METHOD Create : RTS_IEC_HANDLE
  VAR_INPUT
    iAddressFamily : INT;  (* Socket address family *)
    diType : DINT;  (* Socket TYPE *)
    diProtocol : DINT;  (* Socket protocol *)
    pResult : POINTER TO RTS_IEC_RESULT;  (* Pointer to runtime system error code (see CmpErrors.library) *)
  END_VAR
                          // check, for reinitilaization
IF (THIS^.hSocket = RTS_INVALID_HANDLE) THEN
	THIS^.hSocket := SysSocket.SysSockCreate(iAddressFamily, diType, diProtocol, pResult);
	Create := THIS^.hSocket;
ELSE
	Create := RTS_INVALID_HANDLE;
END_IF
                        
END_METHOD
END_FUNCTION_BLOCK

FUNCTION_BLOCK _FB_ETHRx_Message_Unpack
  VAR_INPUT
    I_Byte_0 : BYTE;
    I_Byte_1 : BYTE;
    I_Byte_2 : BYTE;
    I_Byte_3 : BYTE;
    I_Byte_4 : BYTE;
    I_Byte_5 : BYTE;
    I_Byte_6 : BYTE;
    I_Byte_7 : BYTE;
  END_VAR
  VAR_OUTPUT
    S_ER_TmOut : BOOL;  (* Input data endpoints *)
    S_Bit_0 : BOOL;  (* Input data endpoints *)
    S_Bit_1 : BOOL;  (* Input data endpoints *)
    S_Bit_2 : BOOL;  (* Input data endpoints *)
    S_Bit_3 : BOOL;  (* Input data endpoints *)
    S_Bit_4 : BOOL;  (* Input data endpoints *)
    S_Bit_5 : BOOL;  (* Input data endpoints *)
    S_Bit_6 : BOOL;  (* Input data endpoints *)
    S_Bit_7 : BOOL;  (* Input data endpoints *)
    X_Byte_0 : BYTE;  (* Input data endpoints *)
    S_Bit_8 : BOOL;  (* Input data endpoints *)
    S_Bit_9 : BOOL;  (* Input data endpoints *)
    S_Bit_10 : BOOL;  (* Input data endpoints *)
    S_Bit_11 : BOOL;  (* Input data endpoints *)
    S_Bit_12 : BOOL;  (* Input data endpoints *)
    S_Bit_13 : BOOL;  (* Input data endpoints *)
    S_Bit_14 : BOOL;  (* Input data endpoints *)
    S_Bit_15 : BOOL;  (* Input data endpoints *)
    X_Byte_1 : BYTE;  (* Input data endpoints *)
    X_Word_0 : WORD;  (* Input data endpoints *)
    S_Bit_16 : BOOL;  (* Input data endpoints *)
    S_Bit_17 : BOOL;  (* Input data endpoints *)
    S_Bit_18 : BOOL;  (* Input data endpoints *)
    S_Bit_19 : BOOL;  (* Input data endpoints *)
    S_Bit_20 : BOOL;  (* Input data endpoints *)
    S_Bit_21 : BOOL;  (* Input data endpoints *)
    S_Bit_22 : BOOL;  (* Input data endpoints *)
    S_Bit_23 : BOOL;  (* Input data endpoints *)
    X_Byte_2 : BYTE;  (* Input data endpoints *)
    S_Bit_24 : BOOL;  (* Input data endpoints *)
    S_Bit_25 : BOOL;  (* Input data endpoints *)
    S_Bit_26 : BOOL;  (* Input data endpoints *)
    S_Bit_27 : BOOL;  (* Input data endpoints *)
    S_Bit_28 : BOOL;  (* Input data endpoints *)
    S_Bit_29 : BOOL;  (* Input data endpoints *)
    S_Bit_30 : BOOL;  (* Input data endpoints *)
    S_Bit_31 : BOOL;  (* Input data endpoints *)
    X_Byte_3 : BYTE;  (* Input data endpoints *)
    S_Bit_32 : BOOL;  (* Input data endpoints *)
    S_Bit_33 : BOOL;  (* Input data endpoints *)
    S_Bit_34 : BOOL;  (* Input data endpoints *)
    S_Bit_35 : BOOL;  (* Input data endpoints *)
    S_Bit_36 : BOOL;  (* Input data endpoints *)
    S_Bit_37 : BOOL;  (* Input data endpoints *)
    S_Bit_38 : BOOL;  (* Input data endpoints *)
    S_Bit_39 : BOOL;  (* Input data endpoints *)
    X_Byte_4 : BYTE;  (* Input data endpoints *)
    S_Bit_40 : BOOL;  (* Input data endpoints *)
    S_Bit_41 : BOOL;  (* Input data endpoints *)
    S_Bit_42 : BOOL;  (* Input data endpoints *)
    S_Bit_43 : BOOL;  (* Input data endpoints *)
    S_Bit_44 : BOOL;  (* Input data endpoints *)
    S_Bit_45 : BOOL;  (* Input data endpoints *)
    S_Bit_46 : BOOL;  (* Input data endpoints *)
    S_Bit_47 : BOOL;  (* Input data endpoints *)
    X_Byte_5 : BYTE;  (* Input data endpoints *)
    X_Word_2 : WORD;  (* Input data endpoints *)
    S_Bit_48 : BOOL;  (* Input data endpoints *)
    S_Bit_49 : BOOL;  (* Input data endpoints *)
    S_Bit_50 : BOOL;  (* Input data endpoints *)
    S_Bit_51 : BOOL;  (* Input data endpoints *)
    S_Bit_52 : BOOL;  (* Input data endpoints *)
    S_Bit_53 : BOOL;  (* Input data endpoints *)
    S_Bit_54 : BOOL;  (* Input data endpoints *)
    S_Bit_55 : BOOL;  (* Input data endpoints *)
    X_Byte_6 : BYTE;  (* Input data endpoints *)
    S_Bit_56 : BOOL;  (* Input data endpoints *)
    S_Bit_57 : BOOL;  (* Input data endpoints *)
    S_Bit_58 : BOOL;  (* Input data endpoints *)
    S_Bit_59 : BOOL;  (* Input data endpoints *)
    S_Bit_60 : BOOL;  (* Input data endpoints *)
    S_Bit_61 : BOOL;  (* Input data endpoints *)
    S_Bit_62 : BOOL;  (* Input data endpoints *)
    S_Bit_63 : BOOL;  (* Input data endpoints *)
    X_Byte_7 : BYTE;  (* Input data endpoints *)
  END_VAR

                    			X_Byte_0 :=I_Byte_0;			
            X_Byte_1 :=I_Byte_1;
            X_Byte_2 :=I_Byte_2;
            X_Byte_3 :=I_Byte_3;
            X_Byte_4 :=I_Byte_4;
            X_Byte_5 :=I_Byte_5;
			X_Byte_6 :=I_Byte_6;
            X_Byte_7 :=I_Byte_7;
			
			S_Bit_0  := BYTE_TO_BOOL(X_Byte_0 AND 2#00000001);
			S_Bit_1  := BYTE_TO_BOOL(X_Byte_0 AND 2#00000010);
			S_Bit_2  := BYTE_TO_BOOL(X_Byte_0 AND 2#00000100);
			S_Bit_3  := BYTE_TO_BOOL(X_Byte_0 AND 2#00001000);
			S_Bit_4  := BYTE_TO_BOOL(X_Byte_0 AND 2#00010000);
			S_Bit_5  := BYTE_TO_BOOL(X_Byte_0 AND 2#00100000);
			S_Bit_6  := BYTE_TO_BOOL(X_Byte_0 AND 2#01000000);
			S_Bit_7  := BYTE_TO_BOOL(X_Byte_0 AND 2#10000000);
			S_Bit_8  := BYTE_TO_BOOL(X_Byte_1 AND 2#00000001);
			S_Bit_9  := BYTE_TO_BOOL(X_Byte_1 AND 2#00000010);
			S_Bit_10  := BYTE_TO_BOOL(X_Byte_1 AND 2#00000100);
			S_Bit_11  := BYTE_TO_BOOL(X_Byte_1 AND 2#00001000);
			S_Bit_12  := BYTE_TO_BOOL(X_Byte_1 AND 2#00010000);
			S_Bit_13  := BYTE_TO_BOOL(X_Byte_1 AND 2#00100000);
			S_Bit_14  := BYTE_TO_BOOL(X_Byte_1 AND 2#01000000);
			S_Bit_15  := BYTE_TO_BOOL(X_Byte_1 AND 2#10000000);
			S_Bit_16  := BYTE_TO_BOOL(X_Byte_2 AND 2#00000001);
			S_Bit_17  := BYTE_TO_BOOL(X_Byte_2 AND 2#00000010);
			S_Bit_18  := BYTE_TO_BOOL(X_Byte_2 AND 2#00000100);
			S_Bit_19  := BYTE_TO_BOOL(X_Byte_2 AND 2#00001000);
			S_Bit_20  := BYTE_TO_BOOL(X_Byte_2 AND 2#00010000);
			S_Bit_21  := BYTE_TO_BOOL(X_Byte_2 AND 2#00100000);
			S_Bit_22  := BYTE_TO_BOOL(X_Byte_2 AND 2#01000000);
			S_Bit_23  := BYTE_TO_BOOL(X_Byte_2 AND 2#10000000);
			S_Bit_24  := BYTE_TO_BOOL(X_Byte_3 AND 2#00000001);
			S_Bit_25  := BYTE_TO_BOOL(X_Byte_3 AND 2#00000010);
			S_Bit_26  := BYTE_TO_BOOL(X_Byte_3 AND 2#00000100);
			S_Bit_27  := BYTE_TO_BOOL(X_Byte_3 AND 2#00001000);
			S_Bit_28  := BYTE_TO_BOOL(X_Byte_3 AND 2#00010000);
			S_Bit_29  := BYTE_TO_BOOL(X_Byte_3 AND 2#00100000);
			S_Bit_30  := BYTE_TO_BOOL(X_Byte_3 AND 2#01000000);
			S_Bit_31  := BYTE_TO_BOOL(X_Byte_3 AND 2#10000000);
			S_Bit_32  := BYTE_TO_BOOL(X_Byte_4 AND 2#00000001);
			S_Bit_33  := BYTE_TO_BOOL(X_Byte_4 AND 2#00000010);
			S_Bit_34  := BYTE_TO_BOOL(X_Byte_4 AND 2#00000100);
			S_Bit_35  := BYTE_TO_BOOL(X_Byte_4 AND 2#00001000);
			S_Bit_36  := BYTE_TO_BOOL(X_Byte_4 AND 2#00010000);
			S_Bit_37  := BYTE_TO_BOOL(X_Byte_4 AND 2#00100000);
			S_Bit_38  := BYTE_TO_BOOL(X_Byte_4 AND 2#01000000);
			S_Bit_39  := BYTE_TO_BOOL(X_Byte_4 AND 2#10000000);
			S_Bit_40  := BYTE_TO_BOOL(X_Byte_5 AND 2#00000001);
			S_Bit_41  := BYTE_TO_BOOL(X_Byte_5 AND 2#00000010);
			S_Bit_42  := BYTE_TO_BOOL(X_Byte_5 AND 2#00000100);
			S_Bit_43  := BYTE_TO_BOOL(X_Byte_5 AND 2#00001000);
			S_Bit_44  := BYTE_TO_BOOL(X_Byte_5 AND 2#00010000);
			S_Bit_45  := BYTE_TO_BOOL(X_Byte_5 AND 2#00100000);
			S_Bit_46  := BYTE_TO_BOOL(X_Byte_5 AND 2#01000000);
			S_Bit_47  := BYTE_TO_BOOL(X_Byte_5 AND 2#10000000);
			S_Bit_48  := BYTE_TO_BOOL(X_Byte_6 AND 2#00000001);
			S_Bit_49  := BYTE_TO_BOOL(X_Byte_6 AND 2#00000010);
			S_Bit_50  := BYTE_TO_BOOL(X_Byte_6 AND 2#00000100);
			S_Bit_51  := BYTE_TO_BOOL(X_Byte_6 AND 2#00001000);
			S_Bit_52  := BYTE_TO_BOOL(X_Byte_6 AND 2#00010000);
			S_Bit_53  := BYTE_TO_BOOL(X_Byte_6 AND 2#00100000);
			S_Bit_54  := BYTE_TO_BOOL(X_Byte_6 AND 2#01000000);
			S_Bit_55  := BYTE_TO_BOOL(X_Byte_6 AND 2#10000000);
			S_Bit_56  := BYTE_TO_BOOL(X_Byte_7 AND 2#00000001);
			S_Bit_57  := BYTE_TO_BOOL(X_Byte_7 AND 2#00000010);
			S_Bit_58  := BYTE_TO_BOOL(X_Byte_7 AND 2#00000100);
			S_Bit_59  := BYTE_TO_BOOL(X_Byte_7 AND 2#00001000);
			S_Bit_60  := BYTE_TO_BOOL(X_Byte_7 AND 2#00010000);
			S_Bit_61  := BYTE_TO_BOOL(X_Byte_7 AND 2#00100000);
			S_Bit_62  := BYTE_TO_BOOL(X_Byte_7 AND 2#01000000);
			S_Bit_63  := BYTE_TO_BOOL(X_Byte_7 AND 2#10000000);
                  
END_FUNCTION_BLOCK

FUNCTION_BLOCK _FB_ETHTx_Message_Unpack
  VAR_INPUT
    S_Bit_0 : BOOL := FALSE;  (* Message Datas *)
    S_Bit_1 : BOOL := FALSE;  (* Message Datas *)
    S_Bit_2 : BOOL := FALSE;  (* Message Datas *)
    S_Bit_3 : BOOL := FALSE;  (* Message Datas *)
    S_Bit_4 : BOOL := FALSE;  (* Message Datas *)
    S_Bit_5 : BOOL := FALSE;  (* Message Datas *)
    S_Bit_6 : BOOL := FALSE;  (* Message Datas *)
    S_Bit_7 : BOOL := FALSE;  (* Message Datas *)
    X_Byte_0 : BYTE := 16#0;  (* Message Datas *)
    S_Bit_8 : BOOL := FALSE;  (* Message Datas *)
    S_Bit_9 : BOOL := FALSE;  (* Message Datas *)
    S_Bit_10 : BOOL := FALSE;  (* Message Datas *)
    S_Bit_11 : BOOL := FALSE;  (* Message Datas *)
    S_Bit_12 : BOOL := FALSE;  (* Message Datas *)
    S_Bit_13 : BOOL := FALSE;  (* Message Datas *)
    S_Bit_14 : BOOL := FALSE;  (* Message Datas *)
    S_Bit_15 : BOOL := FALSE;  (* Message Datas *)
    X_Byte_1 : BYTE := 16#0;  (* Message Datas *)
    S_Bit_16 : BOOL := FALSE;  (* Message Datas *)
    S_Bit_17 : BOOL := FALSE;  (* Message Datas *)
    S_Bit_18 : BOOL := FALSE;  (* Message Datas *)
    S_Bit_19 : BOOL := FALSE;  (* Message Datas *)
    S_Bit_20 : BOOL := FALSE;  (* Message Datas *)
    S_Bit_21 : BOOL := FALSE;  (* Message Datas *)
    S_Bit_22 : BOOL := FALSE;  (* Message Datas *)
    S_Bit_23 : BOOL := FALSE;  (* Message Datas *)
    X_Byte_2 : BYTE := 16#0;  (* Message Datas *)
    S_Bit_24 : BOOL := FALSE;  (* Message Datas *)
    S_Bit_25 : BOOL := FALSE;  (* Message Datas *)
    S_Bit_26 : BOOL := FALSE;  (* Message Datas *)
    S_Bit_27 : BOOL := FALSE;  (* Message Datas *)
    S_Bit_28 : BOOL := FALSE;  (* Message Datas *)
    S_Bit_29 : BOOL := FALSE;  (* Message Datas *)
    S_Bit_30 : BOOL := FALSE;  (* Message Datas *)
    S_Bit_31 : BOOL := FALSE;  (* Message Datas *)
    X_Byte_3 : BYTE := 16#0;  (* Message Datas *)
    S_Bit_32 : BOOL := FALSE;  (* Message Datas *)
    S_Bit_33 : BOOL := FALSE;  (* Message Datas *)
    S_Bit_34 : BOOL := FALSE;  (* Message Datas *)
    S_Bit_35 : BOOL := FALSE;  (* Message Datas *)
    S_Bit_36 : BOOL := FALSE;  (* Message Datas *)
    S_Bit_37 : BOOL := FALSE;  (* Message Datas *)
    S_Bit_38 : BOOL := FALSE;  (* Message Datas *)
    S_Bit_39 : BOOL := FALSE;  (* Message Datas *)
    X_Byte_4 : BYTE := 16#0;  (* Message Datas *)
    S_Bit_40 : BOOL := FALSE;  (* Message Datas *)
    S_Bit_41 : BOOL := FALSE;  (* Message Datas *)
    S_Bit_42 : BOOL := FALSE;  (* Message Datas *)
    S_Bit_43 : BOOL := FALSE;  (* Message Datas *)
    S_Bit_44 : BOOL := FALSE;  (* Message Datas *)
    S_Bit_45 : BOOL := FALSE;  (* Message Datas *)
    S_Bit_46 : BOOL := FALSE;  (* Message Datas *)
    S_Bit_47 : BOOL := FALSE;  (* Message Datas *)
    X_Byte_5 : BYTE := 16#0;  (* Message Datas *)
    S_Bit_48 : BOOL := FALSE;  (* Message Datas *)
    S_Bit_49 : BOOL := FALSE;  (* Message Datas *)
    S_Bit_50 : BOOL := FALSE;  (* Message Datas *)
    S_Bit_51 : BOOL := FALSE;  (* Message Datas *)
    S_Bit_52 : BOOL := FALSE;  (* Message Datas *)
    S_Bit_53 : BOOL := FALSE;  (* Message Datas *)
    S_Bit_54 : BOOL := FALSE;  (* Message Datas *)
    S_Bit_55 : BOOL := FALSE;  (* Message Datas *)
    X_Byte_6 : BYTE := 16#0;  (* Message Datas *)
    S_Bit_56 : BOOL := FALSE;  (* Message Datas *)
    S_Bit_57 : BOOL := FALSE;  (* Message Datas *)
    S_Bit_58 : BOOL := FALSE;  (* Message Datas *)
    S_Bit_59 : BOOL := FALSE;  (* Message Datas *)
    S_Bit_60 : BOOL := FALSE;  (* Message Datas *)
    S_Bit_61 : BOOL := FALSE;  (* Message Datas *)
    S_Bit_62 : BOOL := FALSE;  (* Message Datas *)
    S_Bit_63 : BOOL := FALSE;  (* Message Datas *)
    X_Byte_7 : BYTE := 16#0;  (* Message Datas *)
  END_VAR
  VAR_OUTPUT
    O_Byte_0 : BYTE;
    O_Byte_1 : BYTE;
    O_Byte_2 : BYTE;
    O_Byte_3 : BYTE;
    O_Byte_4 : BYTE;
    O_Byte_5 : BYTE;
    O_Byte_6 : BYTE;
    O_Byte_7 : BYTE;
  END_VAR
  VAR
    _FB_Pack_Bit_To_Byte_01 : _FB_PACK_8BITS_TO_BYTE;
    _FB_Pack_Bit_To_Byte_02 : _FB_PACK_8BITS_TO_BYTE;
    _FB_Pack_Bit_To_Byte_03 : _FB_PACK_8BITS_TO_BYTE;
    _FB_Pack_Bit_To_Byte_04 : _FB_PACK_8BITS_TO_BYTE;
    _FB_Pack_Bit_To_Byte_05 : _FB_PACK_8BITS_TO_BYTE;
    _FB_Pack_Bit_To_Byte_06 : _FB_PACK_8BITS_TO_BYTE;
    _FB_Pack_Bit_To_Byte_07 : _FB_PACK_8BITS_TO_BYTE;
    _FB_Pack_Bit_To_Byte_08 : _FB_PACK_8BITS_TO_BYTE;
  END_VAR

                    IF X_Byte_0 <> 0 THEN
	
	O_Byte_0 := X_Byte_0;
	
ELSIF S_Bit_0 OR S_Bit_1 OR S_Bit_2 OR S_Bit_3 OR S_Bit_4 OR S_Bit_5 OR S_Bit_6 OR S_Bit_7 THEN			(*Check the bits, pack and assign to the output data*)
	_FB_Pack_Bit_To_Byte_01(
	S_Bit_0:= S_Bit_0, 
	S_Bit_1:= S_Bit_1, 
	S_Bit_2:= S_Bit_2, 
	S_Bit_3:= S_Bit_3, 
	S_Bit_4:= S_Bit_4, 
	S_Bit_5:= S_Bit_5, 
	S_Bit_6:= S_Bit_6, 
	S_Bit_7:= S_Bit_7, 
	X_Byte_0=> O_Byte_0);
ELSE
	O_Byte_0 := 0;
END_IF
		
IF X_Byte_1 <> 0 THEN
	O_Byte_1 := X_Byte_1;
ELSIF S_Bit_8 OR S_Bit_9 OR S_Bit_10 OR S_Bit_11 OR S_Bit_12 OR S_Bit_13 OR S_Bit_14 OR S_Bit_15 THEN			(*Check the bits, pack and assign to the output data*)
	_FB_Pack_Bit_To_Byte_02(
	S_Bit_0:= S_Bit_8, 
	S_Bit_1:= S_Bit_9, 
	S_Bit_2:= S_Bit_10, 
	S_Bit_3:= S_Bit_11, 
	S_Bit_4:= S_Bit_12, 
	S_Bit_5:= S_Bit_13, 
	S_Bit_6:= S_Bit_14, 
	S_Bit_7:= S_Bit_15, 
	X_Byte_0=> O_Byte_1);
ELSE
	O_Byte_1 :=0;
END_IF
	

IF X_Byte_2 <> 0 THEN
	O_Byte_2 := X_Byte_2;
ELSIF S_Bit_16 OR S_Bit_17 OR S_Bit_18 OR S_Bit_19 OR S_Bit_20 OR S_Bit_21 OR S_Bit_22 OR S_Bit_23 THEN				(*Check the bits, pack and assign to the output data*)
	_FB_Pack_Bit_To_Byte_03(
	S_Bit_0:= S_Bit_16, 
	S_Bit_1:= S_Bit_17, 
	S_Bit_2:= S_Bit_18, 
	S_Bit_3:= S_Bit_19, 
	S_Bit_4:= S_Bit_20, 
	S_Bit_5:= S_Bit_21, 
	S_Bit_6:= S_Bit_22, 
	S_Bit_7:= S_Bit_23, 
	X_Byte_0=> O_Byte_2);
ELSE
	O_Byte_2 :=0;
END_IF
		
IF X_Byte_3 <> 0 THEN
	O_Byte_3 := X_Byte_3;
ELSIF S_Bit_24 OR S_Bit_25 OR S_Bit_26 OR S_Bit_27 OR S_Bit_28 OR S_Bit_29 OR S_Bit_30 OR S_Bit_31 THEN				(*Check the bits, pack and assign to the output data*)
	_FB_Pack_Bit_To_Byte_04(
	S_Bit_0:= S_Bit_24, 
	S_Bit_1:= S_Bit_25, 
	S_Bit_2:= S_Bit_26, 
	S_Bit_3:= S_Bit_27, 
	S_Bit_4:= S_Bit_28, 
	S_Bit_5:= S_Bit_29, 
	S_Bit_6:= S_Bit_30, 
	S_Bit_7:= S_Bit_31, 
	X_Byte_0=> O_Byte_3);
ELSE
	O_Byte_3 :=0;
END_IF



IF X_Byte_4 <> 0 THEN
	O_Byte_4 := X_Byte_4;
ELSIF S_Bit_32 OR S_Bit_33 OR S_Bit_34 OR S_Bit_35 OR S_Bit_36 OR S_Bit_37 OR S_Bit_38 OR S_Bit_39 THEN				(*Check the bits, pack and assign to the output data*)
	_FB_Pack_Bit_To_Byte_05(
	S_Bit_0:= S_Bit_32, 
	S_Bit_1:= S_Bit_33, 
	S_Bit_2:= S_Bit_34, 
	S_Bit_3:= S_Bit_35, 
	S_Bit_4:= S_Bit_36, 
	S_Bit_5:= S_Bit_37, 
	S_Bit_6:= S_Bit_38, 
	S_Bit_7:= S_Bit_39, 
	X_Byte_0=> O_Byte_4);	
ELSE
	O_Byte_4 :=0;
END_IF
		
IF X_Byte_5 <> 0 THEN
	O_Byte_5 := X_Byte_5;
ELSIF S_Bit_40 OR S_Bit_41 OR S_Bit_42 OR S_Bit_43 OR S_Bit_44 OR S_Bit_45 OR S_Bit_46 OR S_Bit_47 THEN				(*Check the bits, pack and assign to the output data*)
	_FB_Pack_Bit_To_Byte_06(
	S_Bit_0:= S_Bit_40, 
	S_Bit_1:= S_Bit_41, 
	S_Bit_2:= S_Bit_42, 
	S_Bit_3:= S_Bit_43, 
	S_Bit_4:= S_Bit_44, 
	S_Bit_5:= S_Bit_45, 
	S_Bit_6:= S_Bit_46, 
	S_Bit_7:= S_Bit_47, 
	X_Byte_0=> O_Byte_5);
ELSE
	O_Byte_5 :=0;
END_IF

	

IF X_Byte_6 <> 0 THEN
	O_Byte_6 := X_Byte_6;
ELSIF S_Bit_48 OR S_Bit_49 OR S_Bit_50 OR S_Bit_51 OR S_Bit_52 OR S_Bit_53 OR S_Bit_54 OR S_Bit_55 THEN				(*Check the bits, pack and assign to the output data*)
	_FB_Pack_Bit_To_Byte_07(
	S_Bit_0:= S_Bit_48, 
	S_Bit_1:= S_Bit_49, 
	S_Bit_2:= S_Bit_50, 
	S_Bit_3:= S_Bit_51, 
	S_Bit_4:= S_Bit_52, 
	S_Bit_5:= S_Bit_53, 
	S_Bit_6:= S_Bit_54, 
	S_Bit_7:= S_Bit_55, 
	X_Byte_0=> O_Byte_6);
ELSE
	O_Byte_6 :=0;
END_IF
		
IF X_Byte_7 <> 0 THEN
	O_Byte_7 := X_Byte_7;
ELSIF S_Bit_56 OR S_Bit_57 OR S_Bit_58 OR S_Bit_59 OR S_Bit_60 OR S_Bit_61 OR S_Bit_62 OR S_Bit_63 THEN				(*Check the bits, pack and assign to the output data*)
	_FB_Pack_Bit_To_Byte_08(
	S_Bit_0:= S_Bit_56, 
	S_Bit_1:= S_Bit_57, 
	S_Bit_2:= S_Bit_58, 
	S_Bit_3:= S_Bit_59, 
	S_Bit_4:= S_Bit_60, 
	S_Bit_5:= S_Bit_61, 
	S_Bit_6:= S_Bit_62, 
	S_Bit_7:= S_Bit_63, 
	X_Byte_0=> O_Byte_7);
ELSE
	O_Byte_7 :=0;
END_IF
                  
END_FUNCTION_BLOCK

PROGRAM _ErrorCB_PRG
  VAR
    diag_state : lib500_types.DIAG_STATETYPE := lib500_types.DIAG_STATETYPE.DIAG_STATE_DISABLED;
    watchdog_state : lib500_types.DIAG_WD_STATETYPE := lib500_types.DIAG_WD_STATETYPE.DIAG_WD_STATE_UNKNOWN;
    error : lib500_types.DIAG_ERRORCODE := (error_code := lib500_types.DIAG_ERRORTYPE.DIAG_E_NOERROR, device_num := lib500_types.DIAG_DEVICETYPE.DIAG_DEV_NONE, faulty_value := 0);
    return_code : lib500_types.IO_ERRORTYPE := lib500_types.IO_ERRORTYPE.IO_E_UNKNOWN;
    reaction : lib500_types.DIAG_REACTION := lib500_types.DIAG_REACTION.DIAG_ERR_SAFESTATE;
    call_count : UDINT := 0;
  END_VAR

                    (* get the reason for the error callback *)

return_code := lib500.DIAG_CDS_GetErrorReason(ADR(diag_state), 
                                              ADR(watchdog_state),
                                              ADR(error));
(*											  
IF (error.device_num = lib500_types.DIAG_DEVICETYPE.IO_PIN_175) THEN
	reaction := lib500_types.DIAG_REACTION.DIAG_ERR_DISABLE_SSW2;
	lib500.DIAG_CDS_SetErrorReaction(reaction);
END_IF

IF (error.device_num = lib500_types.DIAG_DEVICETYPE.IO_PIN_153) THEN
	reaction := lib500_types.DIAG_REACTION.DIAG_ERR_DISABLE_SSW0;
	lib500.DIAG_CDS_SetErrorReaction(reaction);
END_IF
IF (error.device_num = lib500_types.DIAG_DEVICETYPE.IO_PIN_101) THEN
	reaction := lib500_types.DIAG_REACTION.DIAG_ERR_DISABLE_SSW2;
	lib500.DIAG_CDS_SetErrorReaction(reaction);
END_IF


IF (error.device_num = lib500_types.DIAG_DEVICETYPE.IO_PIN_155) THEN
	reaction := lib500_types.DIAG_REACTION.DIAG_ERR_SAFESTATE;
	lib500.DIAG_CDS_SetErrorReaction(reaction);
END_IF


*)
(*
IF (error.device_num = lib500_types.DIAG_DEVICETYPE.IO_PIN_177) THEN
	reaction := lib500_types.DIAG_REACTION.DIAG_ERR_DISABLE_SSW0;
	lib500.DIAG_CDS_SetErrorReaction(reaction);
END_IF
*)
(* custom handler code can be placed here *)

(* the choices for the reactions are:
   -> lib500_types.DIAG_REACTION.DIAG_ERR_NOACTION
   -> lib500_types.DIAG_REACTION.DIAG_ERR_SAFESTATE
   -> lib500_types.DIAG_REACTION.DIAG_ERR_DISABLE_SSW0
   -> lib500_types.DIAG_REACTION.DIAG_ERR_DISABLE_SSW1
   -> lib500_types.DIAG_REACTION.DIAG_ERR_DISABLE_SSW2
   -> lib500_types.DIAG_REACTION.DIAG_ERR_DISABLE_HS00
   -> lib500_types.DIAG_REACTION.DIAG_ERR_DISABLE_HS01
   -> lib500_types.DIAG_REACTION.DIAG_ERR_DISABLE_HS02
   -> lib500_types.DIAG_REACTION.DIAG_ERR_DISABLE_HS03
   -> lib500_types.DIAG_REACTION.DIAG_ERR_DISABLE_HS04
   -> lib500_types.DIAG_REACTION.DIAG_ERR_DISABLE_HS05
   -> lib500_types.DIAG_REACTION.DIAG_ERR_DISABLE_HS06
   -> lib500_types.DIAG_REACTION.DIAG_ERR_DISABLE_HS07
   
   it's also possible to combine (binary-or) reactions, like:
   -> lib500_types.DIAG_REACTION.DIAG_ERR_DISABLE_SSW0 OR 
      lib500_types.DIAG_REACTION.DIAG_ERR_DISABLE_SSW1
*)

(* pass the error reaction to the DIAG system *)
lib500.DIAG_CDS_SetErrorReaction(reaction);

(* increment call count *)
call_count := call_count + 1;
                  
END_PROGRAM

PROGRAM _NotificationCB_PRG
  VAR
    diag_state : lib500_types.DIAG_STATETYPE := lib500_types.DIAG_STATETYPE.DIAG_STATE_DISABLED;
    watchdog_state : lib500_types.DIAG_WD_STATETYPE := lib500_types.DIAG_WD_STATETYPE.DIAG_WD_STATE_UNKNOWN;
    error : lib500_types.DIAG_ERRORCODE := (error_code := lib500_types.DIAG_ERRORTYPE.DIAG_E_NOERROR, device_num := lib500_types.DIAG_DEVICETYPE.DIAG_DEV_NONE, faulty_value := 0);
    return_code : lib500_types.IO_ERRORTYPE := lib500_types.IO_ERRORTYPE.IO_E_UNKNOWN;
    call_count : UDINT := 0;
  END_VAR

                    (* get the reason for the notification callback *)
return_code := lib500.DIAG_CDS_GetNotificationReason(ADR(diag_state), 
                                                     ADR(watchdog_state),
                                                     ADR(error));

(* custom handler code can be placed here *)

(* increment call count *)
call_count := call_count + 1;
                  
END_PROGRAM

(* PR1006_REV_002374_TIMTRO, Serdar Temeltaşı @16.05.2025 0x412 mesajına ait extended bilgisi düzeltildi. PR1006_REV_002619_TIMTRO, Serdar Temeltaşı @03.07.2025 0x260, 0x261, 0x262 ve 0x264 mesaj ID'li sinyaller ECU yazılımında düzenlendi. PR1006_REV_002664_TIMTRO, Deniz Çıkış @09.07.2025 VCU'dan alınan DWP parametrelerinin resolution'ı 5 yapıldı. PR1006_REV_002685_TIMTRO, Deniz Çıkış @10.07.2025 DIAG SIS'ten alınan sigorta sinyallerinin byte-bit sıralaması düzeltildi PR1006_REV_002729_TIMTRO, Serdar Temeltaşı @17.07.2025 VCU tarafından gönderilen preheater su tankı seviyesi düşük bilgisi DIAG hattından 0x226 mesajı ile alındı. *)
PROGRAM P_IIVD
  VAR
    _FB_CanRx_Message_500 : _FB_CanRx_Message;  (* Test sürüsü için yapıldı - 22.08.2023 *)
    _FB_CanRx_Message_Unpack_200 : _FB_CanRx_Message_Unpack;
    _FB_CanRx_Message_Unpack_210 : _FB_CanRx_Message_Unpack;
    _FB_CanRx_Message_Unpack_211 : _FB_CanRx_Message_Unpack;
    _FB_CanRx_Message_Unpack_220 : _FB_CanRx_Message_Unpack;
    _FB_CanRx_Message_221 : _FB_CanRx_Message;
    _FB_CanRx_Message_Unpack_222 : _FB_CanRx_Message_Unpack;
    _FB_CanRx_Message_223 : _FB_CanRx_Message;
    _FB_CanRx_Message_224 : _FB_CanRx_Message;
    _FB_CanRx_Message_Unpack_225 : _FB_CanRx_Message_Unpack;
    _FB_CanRx_Message_Unpack_226 : _FB_CanRx_Message_Unpack;
    _FB_CanRx_Message_230 : _FB_CanRx_Message;
    _FB_CanRx_Message_231 : _FB_CanRx_Message;
    _FB_CanRx_Message_232 : _FB_CanRx_Message;
    _FB_CanRx_Message_233 : _FB_CanRx_Message;
    _FB_CanRx_Message_234 : _FB_CanRx_Message;
    _FB_CanRx_Message_Unpack_235 : _FB_CanRx_Message_Unpack;
    _FB_CanRx_Message_Unpack_237 : _FB_CanRx_Message_Unpack;
    _FB_CanRx_Message_Unpack_238 : _FB_CanRx_Message_Unpack;
    _FB_CanRx_Message_Unpack_260 : _FB_CanRx_Message_Unpack;
    _FB_CanRx_Message_Unpack_261 : _FB_CanRx_Message_Unpack;
    _FB_CanRx_Message_Unpack_262 : _FB_CanRx_Message_Unpack;
    _FB_CanRx_Message_Unpack_263 : _FB_CanRx_Message_Unpack;
    _FB_CanRx_Message_Unpack_264 : _FB_CanRx_Message_Unpack;
    _FB_CanRx_Message_Unpack_300 : _FB_CanRx_Message_Unpack;
    _FB_CanRx_Message_Unpack_301 : _FB_CanRx_Message_Unpack;
    _FB_CanRx_Message_Unpack_302 : _FB_CanRx_Message_Unpack;
    _FB_CanRx_Message_Unpack_303 : _FB_CanRx_Message_Unpack;
    _FB_CanRx_Message_Unpack_310 : _FB_CanRx_Message_Unpack;
    _FB_CanRx_Message_Unpack_2E1 : _FB_CanRx_Message_Unpack;
    _FB_CanRx_Message_Unpack_412 : _FB_CanRx_Message_Unpack;
    Raw_W_Str_Pmp_Spd : WORD;
    Raw_X_Str_Pmp_Spd : WORD;
    Raw_X_P_Str_Pmp : WORD;
    Raw_X_I_Str_Pmp : WORD;
    Raw_X_T_Str_Pmp_Mot : BYTE;
    Raw_X_T_Str_Pmp_Inver : BYTE;
    Raw_X_Mot_Load_Str_Pmp : BYTE;
    Raw_X_T_Air_Cmp : BYTE;
    Raw_Z_Config_Clu : BYTE;
    Raw_Z_Ret_Lv : BYTE;
    Raw_X_Axl1_Brk_Ling_1 : BYTE;
    Raw_X_Axl1_Brk_Ling_2 : BYTE;
    Raw_X_Axl2_Brk_Ling_1 : BYTE;
    Raw_X_Axl2_Brk_Ling_2 : BYTE;
    Raw_X_Axl3_Brk_Ling_1 : BYTE;
    Raw_X_Axl3_Brk_Ling_2 : BYTE;
    Raw_X_Axl4_Brk_Ling_1 : BYTE;
    Raw_X_Axl4_Brk_Ling_2 : BYTE;
    Raw_X_Pr_Air_Tank_Brk_Bwd : BYTE;
    Raw_X_Pr_Air_Tank_Brk_Frnt : BYTE;
    Raw_X_Pr_Air_Tank_Brk_Prk : BYTE;
    Raw_X_Pr_Air_Tank_Susp_Rr : BYTE;
    Raw_X_Pr_Air_Tank_Susp_Frnt : BYTE;
    Raw_X_Pr_Axl1_Wh1 : BYTE;
    Raw_X_Pr_Axl1_Wh2 : BYTE;
    Raw_X_Pr_Axl2_Wh1 : BYTE;
    Raw_X_Pr_Axl2_Wh2 : BYTE;
    Raw_X_Pr_Axl2_Wh3 : BYTE;
    Raw_X_Pr_Axl2_Wh4 : BYTE;
    Raw_X_Pr_Axl3_Wh1 : BYTE;
    Raw_X_Pr_Axl3_Wh2 : BYTE;
    Raw_X_Pr_Axl3_Wh3 : BYTE;
    Raw_X_Pr_Axl3_Wh4 : BYTE;
    Raw_X_Pr_Axl4_Wh1 : BYTE;
    Raw_X_Pr_Axl4_Wh2 : BYTE;
    Raw_X_Pr_Axl4_Wh3 : BYTE;
    Raw_X_Pr_Axl4_Wh4 : BYTE;
    Raw_X_Psng_No : BYTE;
    Raw_X_Wgt_Axle : WORD;
    Raw_Z_Dr1_Err_Fram_1 : BYTE;
    Raw_Z_Dr1_Err_Fram_2 : BYTE;
    Raw_Z_Dr1_Err_Fram_3 : BYTE;
    Raw_Z_Dr2_Err_Fram_1 : BYTE;
    Raw_Z_Dr2_Err_Fram_2 : BYTE;
    Raw_Z_Dr2_Err_Fram_3 : BYTE;
    Raw_Z_Dr3_Err_Fram_1 : BYTE;
    Raw_Z_Dr3_Err_Fram_2 : BYTE;
    Raw_Z_Dr3_Err_Fram_3 : BYTE;
    Raw_Z_Dr4_Err_Fram_1 : BYTE;
    Raw_Z_Dr4_Err_Fram_2 : BYTE;
    Raw_Z_Dr4_Err_Fram_3 : BYTE;
    Raw_Z_Dr5_Err_Fram_1 : BYTE;
    Raw_Z_Dr5_Err_Fram_2 : BYTE;
    Raw_Z_Dr5_Err_Fram_3 : BYTE;
    Raw_Z_Dr6_Err_Fram_1 : BYTE;
    Raw_Z_Dr6_Err_Fram_2 : BYTE;
    Raw_Z_Dr6_Err_Fram_3 : BYTE;
    Raw_Z_Dr7_Err_Fram_1 : BYTE;
    Raw_Z_Dr7_Err_Fram_2 : BYTE;
    Raw_Z_Dr7_Err_Fram_3 : BYTE;
    Raw_Z_Dr8_Err_Fram_1 : BYTE;
    Raw_Z_Dr8_Err_Fram_2 : BYTE;
    Raw_Z_Dr8_Err_Fram_3 : BYTE;
    Raw_Z_Dr9_Err_Fram_1 : BYTE;
    Raw_Z_Dr9_Err_Fram_2 : BYTE;
    Raw_Z_Dr9_Err_Fram_3 : BYTE;
    Raw_P_Set_Tm_Dr_Cl_Rls : BYTE;
    Raw_P_Set_Tm_Rout_Pnl_ShtDn : BYTE;
    Raw_P_Set_Tm_Lgt_Dr_ShtDn : BYTE;
    Raw_N_Diag_Lf : BYTE;
    Raw_W_Rd_Par_ID : BYTE;
    Raw_X_Minute : BYTE;
    Raw_X_Hour : BYTE;
    Raw_X_Day : BYTE;
    Raw_X_Month : BYTE;
    Raw_X_Year : BYTE;
    Raw_X_Par_Val : WORD;
    Raw_X_Par_Month : BYTE;
    Raw_X_Par_Year : BYTE;
    Raw_X_Sw_Ver_Mjr_DWP : BYTE;
    Raw_X_Sw_Ver_Mnr_DWP : BYTE;
    Raw_X_Sw_Ver_Tst_DWP : BYTE;
    Raw_X_Sw_Ver_Mjr_VCU : BYTE;
    Raw_X_Sw_Ver_Mnr_VCU : BYTE;
    Raw_X_Sw_Ver_Tst_VCU : BYTE;
    Raw_X_Sw_Ver_Mjr_ATS : BYTE;
    Raw_X_Sw_Ver_Mnr_ATS : BYTE;
    Raw_W_Odo : DWORD;
    Raw_X_Spd_Max : BYTE;
    Raw_X_T_Flr_1 : BYTE;
    Raw_X_T_Flr_2 : BYTE;
    Raw_W_T_Flr : BYTE;
    Raw_X_Fus_0_D1 : BYTE;
    Raw_X_Fus_0_D2 : BYTE;
    Raw_X_Fus_0_D3 : BYTE;
    Raw_X_Fus_0_D4 : BYTE;
    Raw_X_Fus_0_D5 : BYTE;
    Raw_X_Fus_0_D6 : BYTE;
    Raw_X_Fus_0_D7 : BYTE;
    Raw_X_Fus_0_D8 : BYTE;
    Raw_X_Fus_1_D1 : BYTE;
    Raw_X_Fus_1_D2 : BYTE;
    Raw_X_Fus_1_D3 : BYTE;
    Raw_X_Fus_1_D4 : BYTE;
    Raw_X_Fus_1_D5 : BYTE;
    Raw_X_Fus_1_D6 : BYTE;
    Raw_X_Fus_1_D7 : BYTE;
    Raw_X_Fus_1_D8 : BYTE;
    Raw_X_Fus_2_D1 : BYTE;
    Raw_X_Fus_2_D2 : BYTE;
    Raw_X_Fus_2_D3 : BYTE;
    Raw_X_Fus_2_D4 : BYTE;
    Raw_X_Fus_2_D5 : BYTE;
    Raw_X_Fus_2_D6 : BYTE;
    Raw_X_Fus_2_D7 : BYTE;
    Raw_X_Fus_2_D8 : BYTE;
    Raw_X_Fus_3_D1 : BYTE;
    Raw_X_Fus_3_D2 : BYTE;
    Raw_X_Fus_3_D3 : BYTE;
    Raw_X_Fus_3_D4 : BYTE;
    Raw_X_Fus_3_D5 : BYTE;
    Raw_X_Fus_3_D6 : BYTE;
    Raw_X_Fus_3_D7 : BYTE;
    Raw_X_Fus_3_D8 : BYTE;
    _FB_PACK_BYTE_TO_WORD_0 : _FB_PACK_BYTE_TO_WORD;
    _FB_PACK_BYTE_TO_WORD_1 : _FB_PACK_BYTE_TO_WORD;
    _FB_PACK_BYTE_TO_WORD_2 : _FB_PACK_BYTE_TO_WORD;
    _FB_PACK_BYTE_TO_WORD_3 : _FB_PACK_BYTE_TO_WORD;
    _FB_PACK_BYTE_TO_WORD_4 : _FB_PACK_BYTE_TO_WORD;
    _FB_PACK_BYTE_TO_WORD_5 : _FB_PACK_BYTE_TO_WORD;
    _FB_PACK_BYTE_TO_WORD_6 : _FB_PACK_BYTE_TO_WORD;
    _FB_PACK_BYTE_TO_WORD_7 : _FB_PACK_BYTE_TO_WORD;
    _FB_PACK_BYTE_TO_WORD_8 : _FB_PACK_BYTE_TO_WORD;
    _FB_PACK_BYTE_TO_WORD_9 : _FB_PACK_BYTE_TO_WORD;
    _FB_PACK_8BITS_TO_BYTE_0 : _FB_PACK_8BITS_TO_BYTE;
    _FB_PACK_8BITS_TO_BYTE_1 : _FB_PACK_8BITS_TO_BYTE;
    _FB_PACK_8BITS_TO_BYTE_2 : _FB_PACK_8BITS_TO_BYTE;
    _FB_PACK_8BITS_TO_BYTE_3 : _FB_PACK_8BITS_TO_BYTE;
    _FB_PACK_8BITS_TO_BYTE_4 : _FB_PACK_8BITS_TO_BYTE;
    _FB_PACK_8BITS_TO_BYTE_5 : _FB_PACK_8BITS_TO_BYTE;
    _FB_PACK_8BITS_TO_BYTE_6 : _FB_PACK_8BITS_TO_BYTE;
    _FB_PACK_8BITS_TO_BYTE_7 : _FB_PACK_8BITS_TO_BYTE;
    _FB_PACK_8BITS_TO_BYTE_8 : _FB_PACK_8BITS_TO_BYTE;
    _FB_PACK_8BITS_TO_BYTE_9 : _FB_PACK_8BITS_TO_BYTE;
    _FB_PACK_BYTE_TO_DWORD_0 : _FB_PACK_BYTE_TO_DWORD;
  END_VAR

                    (*
**********************************************************************
Bozankaya A.Ş.
**********************************************************************
Name					: P_IIVD_T
POU Type				: Program
Created by              : COMMUNICATION INTERFACE GENERATOR V1.1.034(denizcikispc) , BZK.
Creation Date 			: 2023-06-06T16:56:20
Modifications			: see version description below


Program Description:This program which is created by automatically by communication interface generator 
 handles the RX (INPUT) can messages according to CAN_500_LIB
*********************************************************************

Version 1	
*********************************************************************
Version Description:
- initial version
*********************************************************************
*)
{region " MESSAGE AREA :Haberlesme_Durumlari- ID:200"}

_FB_CanRx_Message_Unpack_200 (	C_Enable	:= GVL.IIVD.S_CAN_Init,
     							Obj_CAN		:= ADR(GVL.IC.Obj_CAN0),
     							X_MsgID		:= 16#200,
     							Tm_MsgTmOut	:= TIME#500MS,
     							S_Extended	:= 0,
     							S_ER_TmOut	=> GVL.IIVD.S_TmOut_Haberlesme_Durumlari_0X200);

{region " SIGNAL AREA : NAME->S_ER_Com_ECU LENGTH->2 STARTBIT :0"}
GVL.IIVD.S_ER_Com_ECU.v					:= NOT GVL.IIVD.S_TmOut_Haberlesme_Durumlari_0X200 AND NOT _FB_CanRx_Message_Unpack_200.S_Bit_1;
GVL.IIVD.S_ER_Com_ECU.x					:= GVL.IIVD.S_ER_Com_ECU.v AND _FB_CanRx_Message_Unpack_200.S_Bit_0;
GVL.IIVD.S_ER_Com_ECU.e					:= _FB_CanRx_Message_Unpack_200.S_Bit_1 AND NOT _FB_CanRx_Message_Unpack_200.S_Bit_0;
GVL.IIVD.S_ER_Com_ECU.na				:= _FB_CanRx_Message_Unpack_200.S_Bit_1 AND _FB_CanRx_Message_Unpack_200.S_Bit_0;
{endregion}
{region " SIGNAL AREA : NAME->S_ER_Com_DWP_ICAN LENGTH->2 STARTBIT :2"}
GVL.IIVD.S_ER_Com_DWP_ICAN.v			:= NOT GVL.IIVD.S_TmOut_Haberlesme_Durumlari_0X200 AND NOT _FB_CanRx_Message_Unpack_200.S_Bit_3;
GVL.IIVD.S_ER_Com_DWP_ICAN.x			:= GVL.IIVD.S_ER_Com_DWP_ICAN.v AND _FB_CanRx_Message_Unpack_200.S_Bit_2;
GVL.IIVD.S_ER_Com_DWP_ICAN.e			:= _FB_CanRx_Message_Unpack_200.S_Bit_3 AND NOT _FB_CanRx_Message_Unpack_200.S_Bit_2;
GVL.IIVD.S_ER_Com_DWP_ICAN.na			:= _FB_CanRx_Message_Unpack_200.S_Bit_3 AND _FB_CanRx_Message_Unpack_200.S_Bit_2;
{endregion}
{region " SIGNAL AREA : NAME->S_ER_Com_DWP_XCAN LENGTH->2 STARTBIT :4"}
GVL.IIVD.S_ER_Com_DWP_XCAN.v			:= NOT GVL.IIVD.S_TmOut_Haberlesme_Durumlari_0X200 AND NOT _FB_CanRx_Message_Unpack_200.S_Bit_5;
GVL.IIVD.S_ER_Com_DWP_XCAN.x			:= GVL.IIVD.S_ER_Com_DWP_XCAN.v AND _FB_CanRx_Message_Unpack_200.S_Bit_4;
GVL.IIVD.S_ER_Com_DWP_XCAN.e			:= _FB_CanRx_Message_Unpack_200.S_Bit_5 AND NOT _FB_CanRx_Message_Unpack_200.S_Bit_4;
GVL.IIVD.S_ER_Com_DWP_XCAN.na			:= _FB_CanRx_Message_Unpack_200.S_Bit_5 AND _FB_CanRx_Message_Unpack_200.S_Bit_4;
{endregion}
{region " SIGNAL AREA : NAME->S_ER_Com_Str_Pmp LENGTH->2 STARTBIT :6"}
GVL.IIVD.S_ER_Com_Str_Pmp.v				:= NOT GVL.IIVD.S_TmOut_Haberlesme_Durumlari_0X200 AND NOT _FB_CanRx_Message_Unpack_200.S_Bit_7;
GVL.IIVD.S_ER_Com_Str_Pmp.x				:= GVL.IIVD.S_ER_Com_Str_Pmp.v AND _FB_CanRx_Message_Unpack_200.S_Bit_6;
GVL.IIVD.S_ER_Com_Str_Pmp.e				:= _FB_CanRx_Message_Unpack_200.S_Bit_7 AND NOT _FB_CanRx_Message_Unpack_200.S_Bit_6;
GVL.IIVD.S_ER_Com_Str_Pmp.na			:= _FB_CanRx_Message_Unpack_200.S_Bit_7 AND _FB_CanRx_Message_Unpack_200.S_Bit_6;
{endregion}
{region " SIGNAL AREA : NAME->S_ER_Com_Fus_Chk_ID0 LENGTH->2 STARTBIT :8"}
GVL.IIVD.S_ER_Com_Fus_Chk_ID0.v			:= NOT GVL.IIVD.S_TmOut_Haberlesme_Durumlari_0X200 AND NOT _FB_CanRx_Message_Unpack_200.S_Bit_9;
GVL.IIVD.S_ER_Com_Fus_Chk_ID0.x			:= GVL.IIVD.S_ER_Com_Fus_Chk_ID0.v AND _FB_CanRx_Message_Unpack_200.S_Bit_8;
GVL.IIVD.S_ER_Com_Fus_Chk_ID0.e			:= _FB_CanRx_Message_Unpack_200.S_Bit_9 AND NOT _FB_CanRx_Message_Unpack_200.S_Bit_8;
GVL.IIVD.S_ER_Com_Fus_Chk_ID0.na		:= _FB_CanRx_Message_Unpack_200.S_Bit_9 AND _FB_CanRx_Message_Unpack_200.S_Bit_8;
{endregion}
{region " SIGNAL AREA : NAME->S_ER_Com_Fus_Chk_ID1 LENGTH->2 STARTBIT :10"}
GVL.IIVD.S_ER_Com_Fus_Chk_ID1.v			:= NOT GVL.IIVD.S_TmOut_Haberlesme_Durumlari_0X200 AND NOT _FB_CanRx_Message_Unpack_200.S_Bit_11;
GVL.IIVD.S_ER_Com_Fus_Chk_ID1.x			:= GVL.IIVD.S_ER_Com_Fus_Chk_ID1.v AND _FB_CanRx_Message_Unpack_200.S_Bit_10;
GVL.IIVD.S_ER_Com_Fus_Chk_ID1.e			:= _FB_CanRx_Message_Unpack_200.S_Bit_11 AND NOT _FB_CanRx_Message_Unpack_200.S_Bit_10;
GVL.IIVD.S_ER_Com_Fus_Chk_ID1.na		:= _FB_CanRx_Message_Unpack_200.S_Bit_11 AND _FB_CanRx_Message_Unpack_200.S_Bit_10;
{endregion}
{region " SIGNAL AREA : NAME->S_ER_Com_Fus_Chk_ID2 LENGTH->2 STARTBIT :12"}
GVL.IIVD.S_ER_Com_Fus_Chk_ID2.v			:= NOT GVL.IIVD.S_TmOut_Haberlesme_Durumlari_0X200 AND NOT _FB_CanRx_Message_Unpack_200.S_Bit_13;
GVL.IIVD.S_ER_Com_Fus_Chk_ID2.x			:= GVL.IIVD.S_ER_Com_Fus_Chk_ID2.v AND _FB_CanRx_Message_Unpack_200.S_Bit_12;
GVL.IIVD.S_ER_Com_Fus_Chk_ID2.e			:= _FB_CanRx_Message_Unpack_200.S_Bit_13 AND NOT _FB_CanRx_Message_Unpack_200.S_Bit_12;
GVL.IIVD.S_ER_Com_Fus_Chk_ID2.na		:= _FB_CanRx_Message_Unpack_200.S_Bit_13 AND _FB_CanRx_Message_Unpack_200.S_Bit_12;
{endregion}
{region " SIGNAL AREA : NAME->S_ER_ECAS LENGTH->2 STARTBIT :14"}
GVL.IIVD.S_ER_Com_ECAS.v				:= NOT GVL.IIVD.S_TmOut_Haberlesme_Durumlari_0X200 AND NOT _FB_CanRx_Message_Unpack_200.S_Bit_15;
GVL.IIVD.S_ER_Com_ECAS.x				:= GVL.IIVD.S_ER_Com_ECAS.v AND _FB_CanRx_Message_Unpack_200.S_Bit_14;
GVL.IIVD.S_ER_Com_ECAS.e				:= _FB_CanRx_Message_Unpack_200.S_Bit_15 AND NOT _FB_CanRx_Message_Unpack_200.S_Bit_14;
GVL.IIVD.S_ER_Com_ECAS.na				:= _FB_CanRx_Message_Unpack_200.S_Bit_15 AND _FB_CanRx_Message_Unpack_200.S_Bit_14;
{endregion}
// PR1006_SRS_000554_TIMTRO
{region " SIGNAL AREA : NAME->S_ER_Com_Snd_Gen LENGTH->2 STARTBIT :16"}
GVL.IIVD.S_ER_Com_Snd_Gen.v				:= NOT GVL.IIVD.S_TmOut_Haberlesme_Durumlari_0X200 AND NOT _FB_CanRx_Message_Unpack_200.S_Bit_17;
GVL.IIVD.S_ER_Com_Snd_Gen.x				:= GVL.IIVD.S_ER_Com_Snd_Gen.v AND _FB_CanRx_Message_Unpack_200.S_Bit_16;
GVL.IIVD.S_ER_Com_Snd_Gen.e				:= _FB_CanRx_Message_Unpack_200.S_Bit_17 AND NOT _FB_CanRx_Message_Unpack_200.S_Bit_16;
GVL.IIVD.S_ER_Com_Snd_Gen.na			:= _FB_CanRx_Message_Unpack_200.S_Bit_17 AND _FB_CanRx_Message_Unpack_200.S_Bit_16;
{endregion}
{region " SIGNAL AREA : NAME->S_ER_Com_DCAN LENGTH->2 STARTBIT :18"}
GVL.IIVD.S_ER_Com_DCAN.v				:= NOT GVL.IIVD.S_TmOut_Haberlesme_Durumlari_0X200 AND NOT _FB_CanRx_Message_Unpack_200.S_Bit_19;
GVL.IIVD.S_ER_Com_DCAN.x				:= GVL.IIVD.S_ER_Com_DCAN.v AND _FB_CanRx_Message_Unpack_200.S_Bit_18;
GVL.IIVD.S_ER_Com_DCAN.e				:= _FB_CanRx_Message_Unpack_200.S_Bit_19 AND NOT _FB_CanRx_Message_Unpack_200.S_Bit_18;
GVL.IIVD.S_ER_Com_DCAN.na				:= _FB_CanRx_Message_Unpack_200.S_Bit_19 AND _FB_CanRx_Message_Unpack_200.S_Bit_18;
{endregion}
{region " SIGNAL AREA : NAME->S_ER_Com_Node1 LENGTH->2 STARTBIT :24"}
GVL.IIVD.S_ER_Com_Node1.v				:= NOT GVL.IIVD.S_TmOut_Haberlesme_Durumlari_0X200 AND NOT _FB_CanRx_Message_Unpack_200.S_Bit_25;
GVL.IIVD.S_ER_Com_Node1.x				:= GVL.IIVD.S_ER_Com_Node1.v AND _FB_CanRx_Message_Unpack_200.S_Bit_24;
GVL.IIVD.S_ER_Com_Node1.e				:= _FB_CanRx_Message_Unpack_200.S_Bit_25 AND NOT _FB_CanRx_Message_Unpack_200.S_Bit_24;
GVL.IIVD.S_ER_Com_Node1.na				:= _FB_CanRx_Message_Unpack_200.S_Bit_25 AND _FB_CanRx_Message_Unpack_200.S_Bit_24;
{endregion}
{region " SIGNAL AREA : NAME->S_ER_Com_Node2 LENGTH->2 STARTBIT :26"}
GVL.IIVD.S_ER_Com_Node2.v				:= NOT GVL.IIVD.S_TmOut_Haberlesme_Durumlari_0X200 AND NOT _FB_CanRx_Message_Unpack_200.S_Bit_27;
GVL.IIVD.S_ER_Com_Node2.x				:= GVL.IIVD.S_ER_Com_Node2.v AND _FB_CanRx_Message_Unpack_200.S_Bit_26;
GVL.IIVD.S_ER_Com_Node2.e				:= _FB_CanRx_Message_Unpack_200.S_Bit_27 AND NOT _FB_CanRx_Message_Unpack_200.S_Bit_26;
GVL.IIVD.S_ER_Com_Node2.na				:= _FB_CanRx_Message_Unpack_200.S_Bit_27 AND _FB_CanRx_Message_Unpack_200.S_Bit_26;
{endregion}
{region " SIGNAL AREA : NAME->S_ER_Com_Node3 LENGTH->2 STARTBIT :28"}
GVL.IIVD.S_ER_Com_Node3.v				:= NOT GVL.IIVD.S_TmOut_Haberlesme_Durumlari_0X200 AND NOT _FB_CanRx_Message_Unpack_200.S_Bit_29;
GVL.IIVD.S_ER_Com_Node3.x				:= GVL.IIVD.S_ER_Com_Node3.v AND _FB_CanRx_Message_Unpack_200.S_Bit_28;
GVL.IIVD.S_ER_Com_Node3.e				:= _FB_CanRx_Message_Unpack_200.S_Bit_29 AND NOT _FB_CanRx_Message_Unpack_200.S_Bit_28;
GVL.IIVD.S_ER_Com_Node3.na				:= _FB_CanRx_Message_Unpack_200.S_Bit_29 AND _FB_CanRx_Message_Unpack_200.S_Bit_28;
{endregion}
{region " SIGNAL AREA : NAME->S_ER_Com_Node4 LENGTH->2 STARTBIT :30"}
GVL.IIVD.S_ER_Com_Node4.v				:= NOT GVL.IIVD.S_TmOut_Haberlesme_Durumlari_0X200 AND NOT _FB_CanRx_Message_Unpack_200.S_Bit_31;
GVL.IIVD.S_ER_Com_Node4.x				:= GVL.IIVD.S_ER_Com_Node4.v AND _FB_CanRx_Message_Unpack_200.S_Bit_30;
GVL.IIVD.S_ER_Com_Node4.e				:= _FB_CanRx_Message_Unpack_200.S_Bit_31 AND NOT _FB_CanRx_Message_Unpack_200.S_Bit_30;
GVL.IIVD.S_ER_Com_Node4.na				:= _FB_CanRx_Message_Unpack_200.S_Bit_31 AND _FB_CanRx_Message_Unpack_200.S_Bit_30;
{endregion}
{region " SIGNAL AREA : NAME->S_ER_Com_Node5 LENGTH->2 STARTBIT :32"}
GVL.IIVD.S_ER_Com_Node5.v				:= NOT GVL.IIVD.S_TmOut_Haberlesme_Durumlari_0X200 AND NOT _FB_CanRx_Message_Unpack_200.S_Bit_33;
GVL.IIVD.S_ER_Com_Node5.x				:= GVL.IIVD.S_ER_Com_Node5.v AND _FB_CanRx_Message_Unpack_200.S_Bit_32;
GVL.IIVD.S_ER_Com_Node5.e				:= _FB_CanRx_Message_Unpack_200.S_Bit_33 AND NOT _FB_CanRx_Message_Unpack_200.S_Bit_32;
GVL.IIVD.S_ER_Com_Node5.na				:= _FB_CanRx_Message_Unpack_200.S_Bit_33 AND _FB_CanRx_Message_Unpack_200.S_Bit_32;
{endregion}
{region " SIGNAL AREA : NAME->S_ER_Com_Node6 LENGTH->2 STARTBIT :34"}
GVL.IIVD.S_ER_Com_Node6.v				:= NOT GVL.IIVD.S_TmOut_Haberlesme_Durumlari_0X200 AND NOT _FB_CanRx_Message_Unpack_200.S_Bit_35;
GVL.IIVD.S_ER_Com_Node6.x				:= GVL.IIVD.S_ER_Com_Node6.v AND _FB_CanRx_Message_Unpack_200.S_Bit_34;
GVL.IIVD.S_ER_Com_Node6.e				:= _FB_CanRx_Message_Unpack_200.S_Bit_35 AND NOT _FB_CanRx_Message_Unpack_200.S_Bit_34;
GVL.IIVD.S_ER_Com_Node6.na				:= _FB_CanRx_Message_Unpack_200.S_Bit_35 AND _FB_CanRx_Message_Unpack_200.S_Bit_34;
{endregion}
{region " SIGNAL AREA : NAME->S_ER_Com_Node5 LENGTH->2 STARTBIT :38"}
GVL.IIVD.S_ER_Com_Node8.v				:= NOT GVL.IIVD.S_TmOut_Haberlesme_Durumlari_0X200 AND NOT _FB_CanRx_Message_Unpack_200.S_Bit_39;
GVL.IIVD.S_ER_Com_Node8.x				:= GVL.IIVD.S_ER_Com_Node8.v AND _FB_CanRx_Message_Unpack_200.S_Bit_38;
GVL.IIVD.S_ER_Com_Node8.e				:= _FB_CanRx_Message_Unpack_200.S_Bit_39 AND NOT _FB_CanRx_Message_Unpack_200.S_Bit_38;
GVL.IIVD.S_ER_Com_Node8.na				:= _FB_CanRx_Message_Unpack_200.S_Bit_39 AND _FB_CanRx_Message_Unpack_200.S_Bit_38;
{endregion}
{region " SIGNAL AREA : NAME->S_ER_Com_Dr1 LENGTH->2 STARTBIT :40"}
GVL.IIVD.S_ER_Com_Dr1.v					:= NOT GVL.IIVD.S_TmOut_Haberlesme_Durumlari_0X200 AND NOT _FB_CanRx_Message_Unpack_200.S_Bit_41;
GVL.IIVD.S_ER_Com_Dr1.x					:= GVL.IIVD.S_ER_Com_Dr1.v AND _FB_CanRx_Message_Unpack_200.S_Bit_40;
GVL.IIVD.S_ER_Com_Dr1.e					:= _FB_CanRx_Message_Unpack_200.S_Bit_41 AND NOT _FB_CanRx_Message_Unpack_200.S_Bit_40;
GVL.IIVD.S_ER_Com_Dr1.na				:= _FB_CanRx_Message_Unpack_200.S_Bit_41 AND _FB_CanRx_Message_Unpack_200.S_Bit_40;
{endregion}
{region " SIGNAL AREA : NAME->S_ER_Com_Dr2 LENGTH->2 STARTBIT :42"}
GVL.IIVD.S_ER_Com_Dr2.v					:= NOT GVL.IIVD.S_TmOut_Haberlesme_Durumlari_0X200 AND NOT _FB_CanRx_Message_Unpack_200.S_Bit_43;
GVL.IIVD.S_ER_Com_Dr2.x					:= GVL.IIVD.S_ER_Com_Dr2.v AND _FB_CanRx_Message_Unpack_200.S_Bit_42;
GVL.IIVD.S_ER_Com_Dr2.e					:= _FB_CanRx_Message_Unpack_200.S_Bit_43 AND NOT _FB_CanRx_Message_Unpack_200.S_Bit_42;
GVL.IIVD.S_ER_Com_Dr2.na				:= _FB_CanRx_Message_Unpack_200.S_Bit_43 AND _FB_CanRx_Message_Unpack_200.S_Bit_42;
{endregion}
{region " SIGNAL AREA : NAME->S_ER_Com_Dr3 LENGTH->2 STARTBIT :44"}
GVL.IIVD.S_ER_Com_Dr3.v					:= NOT GVL.IIVD.S_TmOut_Haberlesme_Durumlari_0X200 AND NOT _FB_CanRx_Message_Unpack_200.S_Bit_45;
GVL.IIVD.S_ER_Com_Dr3.x					:= GVL.IIVD.S_ER_Com_Dr3.v AND _FB_CanRx_Message_Unpack_200.S_Bit_44;
GVL.IIVD.S_ER_Com_Dr3.e					:= _FB_CanRx_Message_Unpack_200.S_Bit_45 AND NOT _FB_CanRx_Message_Unpack_200.S_Bit_44;
GVL.IIVD.S_ER_Com_Dr3.na				:= _FB_CanRx_Message_Unpack_200.S_Bit_45 AND _FB_CanRx_Message_Unpack_200.S_Bit_44;
{endregion}
{region " SIGNAL AREA : NAME->S_ER_Com_Dr4 LENGTH->2 STARTBIT :46"}
GVL.IIVD.S_ER_Com_Dr4.v					:= NOT GVL.IIVD.S_TmOut_Haberlesme_Durumlari_0X200 AND NOT _FB_CanRx_Message_Unpack_200.S_Bit_47;
GVL.IIVD.S_ER_Com_Dr4.x					:= GVL.IIVD.S_ER_Com_Dr4.v AND _FB_CanRx_Message_Unpack_200.S_Bit_46;
GVL.IIVD.S_ER_Com_Dr4.e					:= _FB_CanRx_Message_Unpack_200.S_Bit_47 AND NOT _FB_CanRx_Message_Unpack_200.S_Bit_46;
GVL.IIVD.S_ER_Com_Dr4.na				:= _FB_CanRx_Message_Unpack_200.S_Bit_47 AND _FB_CanRx_Message_Unpack_200.S_Bit_46;
{endregion}
{region " SIGNAL AREA : NAME->S_ER_Com_Dr5 LENGTH->2 STARTBIT :48"}
GVL.IIVD.S_ER_Com_Dr5.v					:= NOT GVL.IIVD.S_TmOut_Haberlesme_Durumlari_0X200 AND NOT _FB_CanRx_Message_Unpack_200.S_Bit_49;
GVL.IIVD.S_ER_Com_Dr5.x					:= GVL.IIVD.S_ER_Com_Dr5.v AND _FB_CanRx_Message_Unpack_200.S_Bit_48;
GVL.IIVD.S_ER_Com_Dr5.e					:= _FB_CanRx_Message_Unpack_200.S_Bit_49 AND NOT _FB_CanRx_Message_Unpack_200.S_Bit_48;
GVL.IIVD.S_ER_Com_Dr5.na				:= _FB_CanRx_Message_Unpack_200.S_Bit_49 AND _FB_CanRx_Message_Unpack_200.S_Bit_48;
{endregion}
{region " SIGNAL AREA : NAME->S_ER_Com_Dr6 LENGTH->2 STARTBIT :50"}
GVL.IIVD.S_ER_Com_Dr6.v					:= NOT GVL.IIVD.S_TmOut_Haberlesme_Durumlari_0X200 AND NOT _FB_CanRx_Message_Unpack_200.S_Bit_51;
GVL.IIVD.S_ER_Com_Dr6.x					:= GVL.IIVD.S_ER_Com_Dr6.v AND _FB_CanRx_Message_Unpack_200.S_Bit_50;
GVL.IIVD.S_ER_Com_Dr6.e					:= _FB_CanRx_Message_Unpack_200.S_Bit_51 AND NOT _FB_CanRx_Message_Unpack_200.S_Bit_50;
GVL.IIVD.S_ER_Com_Dr6.na				:= _FB_CanRx_Message_Unpack_200.S_Bit_51 AND _FB_CanRx_Message_Unpack_200.S_Bit_50;
{endregion}
{region " SIGNAL AREA : NAME->S_ER_Com_Dr7 LENGTH->2 STARTBIT :52"}
GVL.IIVD.S_ER_Com_Dr7.v					:= NOT GVL.IIVD.S_TmOut_Haberlesme_Durumlari_0X200 AND NOT _FB_CanRx_Message_Unpack_200.S_Bit_53;
GVL.IIVD.S_ER_Com_Dr7.x					:= GVL.IIVD.S_ER_Com_Dr7.v AND _FB_CanRx_Message_Unpack_200.S_Bit_52;
GVL.IIVD.S_ER_Com_Dr7.e					:= _FB_CanRx_Message_Unpack_200.S_Bit_53 AND NOT _FB_CanRx_Message_Unpack_200.S_Bit_52;
GVL.IIVD.S_ER_Com_Dr7.na				:= _FB_CanRx_Message_Unpack_200.S_Bit_53 AND _FB_CanRx_Message_Unpack_200.S_Bit_52;
{endregion}
{region " SIGNAL AREA : NAME->S_ER_Com_Dr8 LENGTH->2 STARTBIT :54"}
GVL.IIVD.S_ER_Com_Dr8.v					:= NOT GVL.IIVD.S_TmOut_Haberlesme_Durumlari_0X200 AND NOT _FB_CanRx_Message_Unpack_200.S_Bit_55;
GVL.IIVD.S_ER_Com_Dr8.x					:= GVL.IIVD.S_ER_Com_Dr8.v AND _FB_CanRx_Message_Unpack_200.S_Bit_54;
GVL.IIVD.S_ER_Com_Dr8.e					:= _FB_CanRx_Message_Unpack_200.S_Bit_55 AND NOT _FB_CanRx_Message_Unpack_200.S_Bit_54;
GVL.IIVD.S_ER_Com_Dr8.na				:= _FB_CanRx_Message_Unpack_200.S_Bit_55 AND _FB_CanRx_Message_Unpack_200.S_Bit_54;
{endregion}
{region " SIGNAL AREA : NAME->S_ER_Com_Dr9 LENGTH->2 STARTBIT :56"}
GVL.IIVD.S_ER_Com_Dr9.v					:= NOT GVL.IIVD.S_TmOut_Haberlesme_Durumlari_0X200 AND NOT _FB_CanRx_Message_Unpack_200.S_Bit_57;
GVL.IIVD.S_ER_Com_Dr9.x					:= GVL.IIVD.S_ER_Com_Dr9.v AND _FB_CanRx_Message_Unpack_200.S_Bit_56;
GVL.IIVD.S_ER_Com_Dr9.e					:= _FB_CanRx_Message_Unpack_200.S_Bit_57 AND NOT _FB_CanRx_Message_Unpack_200.S_Bit_56;
GVL.IIVD.S_ER_Com_Dr9.na				:= _FB_CanRx_Message_Unpack_200.S_Bit_57 AND _FB_CanRx_Message_Unpack_200.S_Bit_56;
{endregion}
// PR1006_SRS_000700_TIMTRO
{region " SIGNAL AREA : NAME->S_Warn_Knl_Mn_Cond LENGTH->2 STARTBIT :58"}
GVL.IIVD.S_Warn_Knl_Mn_Cond.v			:= NOT GVL.IIVD.S_TmOut_Haberlesme_Durumlari_0X200 AND NOT _FB_CanRx_Message_Unpack_200.S_Bit_59;
GVL.IIVD.S_Warn_Knl_Mn_Cond.x 			:= GVL.IIVD.S_Warn_Knl_Mn_Cond.v AND _FB_CanRx_Message_Unpack_200.S_Bit_58;
GVL.IIVD.S_Warn_Knl_Mn_Cond.e			:= _FB_CanRx_Message_Unpack_200.S_Bit_59 AND NOT _FB_CanRx_Message_Unpack_200.S_Bit_58;
GVL.IIVD.S_Warn_Knl_Mn_Cond.na			:= _FB_CanRx_Message_Unpack_200.S_Bit_59 AND _FB_CanRx_Message_Unpack_200.S_Bit_58;
{endregion}
// PR1006_SRS_000799_TIMTRO
{region " SIGNAL AREA : NAME->S_ER_Lmp_Oc LENGTH->2 STARTBIT :60"}
GVL.IIVD.S_ER_Lmp_Oc.v					:= NOT GVL.IIVD.S_TmOut_Haberlesme_Durumlari_0X200 AND NOT _FB_CanRx_Message_Unpack_200.S_Bit_61;
GVL.IIVD.S_ER_Lmp_Oc.x 					:= GVL.IIVD.S_ER_Lmp_Oc.v AND _FB_CanRx_Message_Unpack_200.S_Bit_60;
GVL.IIVD.S_ER_Lmp_Oc.e					:= _FB_CanRx_Message_Unpack_200.S_Bit_61 AND NOT _FB_CanRx_Message_Unpack_200.S_Bit_60;
GVL.IIVD.S_ER_Lmp_Oc.na					:= _FB_CanRx_Message_Unpack_200.S_Bit_61 AND _FB_CanRx_Message_Unpack_200.S_Bit_60;
{endregion}
// PR1006_SRS_001017_TIMTRO
{region " SIGNAL AREA : NAME->S_ER_Lmp_Oc LENGTH->2 STARTBIT :62"}
GVL.IIVD.S_ER_Mir_Windw_Heat_En.v		:= NOT GVL.IIVD.S_TmOut_Haberlesme_Durumlari_0X200 AND NOT _FB_CanRx_Message_Unpack_200.S_Bit_63;
GVL.IIVD.S_ER_Mir_Windw_Heat_En.x 		:= GVL.IIVD.S_ER_Mir_Windw_Heat_En.v AND _FB_CanRx_Message_Unpack_200.S_Bit_62;
GVL.IIVD.S_ER_Mir_Windw_Heat_En.e		:= _FB_CanRx_Message_Unpack_200.S_Bit_63 AND NOT _FB_CanRx_Message_Unpack_200.S_Bit_62;
GVL.IIVD.S_ER_Mir_Windw_Heat_En.na		:= _FB_CanRx_Message_Unpack_200.S_Bit_63 AND _FB_CanRx_Message_Unpack_200.S_Bit_62;
{endregion}
{endregion}

{region " MESSAGE AREA :Direksiyon_Pompasi_Analog- ID:210"}

_FB_CanRx_Message_Unpack_210 (	C_Enable	:= GVL.IIVD.S_CAN_Init,
     							Obj_CAN		:= ADR(GVL.IC.Obj_CAN0),
     							X_MsgID		:= 16#210,
     							Tm_MsgTmOut	:= TIME#2500MS,
     							S_Extended	:= 0,
     							S_ER_TmOut	=> GVL.IIVD.S_TmOut_Direksiyon_Pompasi_Analog_0X210);

{region " SIGNAL AREA : NAME->W_Str_Pmp_Spd LENGTH->16 STARTBIT :0"}
_FB_PACK_BYTE_TO_WORD_0 (	X_BYTE_0	:= _FB_CanRx_Message_Unpack_210.X_Byte_0, 
							X_BYTE_1	:=  _FB_CanRx_Message_Unpack_210.X_Byte_1, 
							X_WORD_0 	=> Raw_W_Str_Pmp_Spd);
GVL.IIVD.W_Str_Pmp_Spd.e				:= (Raw_W_Str_Pmp_Spd > 16#FDFF) AND (Raw_W_Str_Pmp_Spd <= 16#FEFF);
GVL.IIVD.W_Str_Pmp_Spd.na				:= (Raw_W_Str_Pmp_Spd > 16#FEFF);
GVL.IIVD.W_Str_Pmp_Spd.RangeExcd		:= NOT ((UINT_TO_REAL(WORD_TO_UINT(Raw_W_Str_Pmp_Spd)) >= 0) AND (UINT_TO_REAL(WORD_TO_UINT(Raw_W_Str_Pmp_Spd)) <= 8000));
GVL.IIVD.W_Str_Pmp_Spd.v				:= NOT( GVL.IIVD.S_TmOut_Direksiyon_Pompasi_Analog_0X210 OR GVL.IIVD.W_Str_Pmp_Spd.RangeExcd OR GVL.IIVD.W_Str_Pmp_Spd.e OR GVL.IIVD.W_Str_Pmp_Spd.na) ;
GVL.IIVD.W_Str_Pmp_Spd.x				:= 
(*SELECT 1 : Is data valid ?*)				SEL(GVL.IIVD.W_Str_Pmp_Spd.v,
(*DEFAULT value assigment*)					0,
(*Transmission is VALID*)					UINT_TO_REAL(WORD_TO_UINT(Raw_W_Str_Pmp_Spd)));
{endregion}
{region " SIGNAL AREA : NAME->X_Str_Pmp_Spd LENGTH->16 STARTBIT :16"}
_FB_PACK_BYTE_TO_WORD_1 (	X_BYTE_0	:= _FB_CanRx_Message_Unpack_210.X_Byte_2, 
							X_BYTE_1	:= _FB_CanRx_Message_Unpack_210.X_Byte_3, 
							X_WORD_0 	=> Raw_X_Str_Pmp_Spd);
GVL.IIVD.X_Str_Pmp_Spd.e				:= (Raw_X_Str_Pmp_Spd > 16#FDFF) AND (Raw_X_Str_Pmp_Spd <= 16#FEFF);
GVL.IIVD.X_Str_Pmp_Spd.na				:= (Raw_X_Str_Pmp_Spd > 16#FEFF);
GVL.IIVD.X_Str_Pmp_Spd.RangeExcd		:= NOT ((UINT_TO_REAL(WORD_TO_UINT(Raw_X_Str_Pmp_Spd)) >= 0) AND (UINT_TO_REAL(WORD_TO_UINT(Raw_X_Str_Pmp_Spd)) <= 8000));
GVL.IIVD.X_Str_Pmp_Spd.v				:= NOT( GVL.IIVD.S_TmOut_Direksiyon_Pompasi_Analog_0X210 OR GVL.IIVD.X_Str_Pmp_Spd.RangeExcd OR GVL.IIVD.X_Str_Pmp_Spd.e OR GVL.IIVD.X_Str_Pmp_Spd.na) ;
GVL.IIVD.X_Str_Pmp_Spd.x				:= 
(*SELECT 1 : Is data valid ?*)				SEL(GVL.IIVD.X_Str_Pmp_Spd.v,
(*DEFAULT value assigment*)					0,
(*Transmission is VALID*)					UINT_TO_REAL(WORD_TO_UINT(Raw_X_Str_Pmp_Spd)));
{endregion}
{region " SIGNAL AREA : NAME->X_P_Str_Pmp LENGTH->16 STARTBIT :32"}
_FB_PACK_BYTE_TO_WORD_2 (	X_BYTE_0	:= _FB_CanRx_Message_Unpack_210.X_Byte_4, 
							X_BYTE_1	:= _FB_CanRx_Message_Unpack_210.X_Byte_5, 
							X_WORD_0 	=> Raw_X_P_Str_Pmp);
GVL.IIVD.X_P_Str_Pmp.e					:= (Raw_X_P_Str_Pmp > 16#FDFF) AND (Raw_X_P_Str_Pmp <= 16#FEFF);
GVL.IIVD.X_P_Str_Pmp.na					:= (Raw_X_P_Str_Pmp > 16#FEFF);
GVL.IIVD.X_P_Str_Pmp.RangeExcd			:= NOT ((UINT_TO_REAL(WORD_TO_UINT(Raw_X_P_Str_Pmp)) >= 0) AND (UINT_TO_REAL(WORD_TO_UINT(Raw_X_P_Str_Pmp)) <= 65000));
GVL.IIVD.X_P_Str_Pmp.v					:= NOT( GVL.IIVD.S_TmOut_Direksiyon_Pompasi_Analog_0X210 OR GVL.IIVD.X_P_Str_Pmp.RangeExcd OR GVL.IIVD.X_P_Str_Pmp.e OR GVL.IIVD.X_P_Str_Pmp.na) ;
GVL.IIVD.X_P_Str_Pmp.x					:= 
(*SELECT 1 : Is data valid ?*)				SEL(GVL.IIVD.X_P_Str_Pmp.v,
(*DEFAULT value assigment*)					0,
(*Transmission is VALID*)					UINT_TO_REAL(WORD_TO_UINT(Raw_X_P_Str_Pmp)));
{endregion}
{region " SIGNAL AREA : NAME->X_I_Str_Pmp LENGTH->9 STARTBIT :48"}
_FB_PACK_BYTE_TO_WORD_3();
_FB_PACK_8BITS_TO_BYTE_0 (	S_BIT_0		:= _FB_CanRx_Message_Unpack_210.S_Bit_48,
							S_BIT_1		:= _FB_CanRx_Message_Unpack_210.S_Bit_49,
							S_BIT_2		:= _FB_CanRx_Message_Unpack_210.S_Bit_50,
							S_BIT_3		:= _FB_CanRx_Message_Unpack_210.S_Bit_51,
							S_BIT_4		:= _FB_CanRx_Message_Unpack_210.S_Bit_52,
							S_BIT_5		:= _FB_CanRx_Message_Unpack_210.S_Bit_53,
							S_BIT_6		:= _FB_CanRx_Message_Unpack_210.S_Bit_54,
							S_BIT_7		:= _FB_CanRx_Message_Unpack_210.S_Bit_55,
							X_BYTE_0	=>_FB_PACK_BYTE_TO_WORD_3.X_BYTE_0);
_FB_PACK_8BITS_TO_BYTE_1 (	S_BIT_0		:= _FB_CanRx_Message_Unpack_210.S_Bit_56 ,
							X_BYTE_0	=>_FB_PACK_BYTE_TO_WORD_3.X_BYTE_1);
Raw_X_I_Str_Pmp            				:=_FB_PACK_BYTE_TO_WORD_3.X_WORD_0;
GVL.IIVD.X_I_Str_Pmp.RangeExcd			:= NOT ((UINT_TO_REAL(WORD_TO_UINT(Raw_X_I_Str_Pmp)) >= 0) AND (UINT_TO_REAL(WORD_TO_UINT(Raw_X_I_Str_Pmp)) <= 511));
GVL.IIVD.X_I_Str_Pmp.v					:= NOT( GVL.IIVD.S_TmOut_Direksiyon_Pompasi_Analog_0X210 OR GVL.IIVD.X_I_Str_Pmp.RangeExcd ) ;
GVL.IIVD.X_I_Str_Pmp.x					:= 
(*SELECT 1 : Is data valid ?*)				SEL(GVL.IIVD.X_I_Str_Pmp.v,
(*DEFAULT value assigment*)					0,
(*Transmission is VALID*)					UINT_TO_REAL(WORD_TO_UINT(Raw_X_I_Str_Pmp)));
{endregion}
{endregion}

{region " MESSAGE AREA :Direksiyon_Pompasi_Durum- ID:211"}

_FB_CanRx_Message_Unpack_211 (	C_Enable	:= GVL.IIVD.S_CAN_Init,
     							Obj_CAN		:= ADR(GVL.IC.Obj_CAN0),
     							X_MsgID		:= 16#211,
     							Tm_MsgTmOut	:= TIME#2500MS,
     							S_Extended	:= 0,
     							S_ER_TmOut	=> GVL.IIVD.S_TmOut_Direksiyon_Pompasi_Durum_0X211);

{region " SIGNAL AREA : NAME->C_Str_Pmp_En LENGTH->2 STARTBIT :0"}
GVL.IIVD.C_Str_Pmp_En.v					:= NOT GVL.IIVD.S_TmOut_Direksiyon_Pompasi_Durum_0X211 AND NOT _FB_CanRx_Message_Unpack_211.S_Bit_1;
GVL.IIVD.C_Str_Pmp_En.x					:= GVL.IIVD.C_Str_Pmp_En.v AND _FB_CanRx_Message_Unpack_211.S_Bit_0;
GVL.IIVD.C_Str_Pmp_En.e					:= _FB_CanRx_Message_Unpack_211.S_Bit_1 AND NOT _FB_CanRx_Message_Unpack_211.S_Bit_0 ;
GVL.IIVD.C_Str_Pmp_En.na				:= _FB_CanRx_Message_Unpack_211.S_Bit_1 AND _FB_CanRx_Message_Unpack_211.S_Bit_0 ;
{endregion}
{region " SIGNAL AREA : NAME->S_Str_Pmp_Em_Run_FOC LENGTH->2 STARTBIT :2"}
GVL.IIVD.S_Str_Pmp_Em_Run_FOC.v			:= NOT GVL.IIVD.S_TmOut_Direksiyon_Pompasi_Durum_0X211 AND NOT _FB_CanRx_Message_Unpack_211.S_Bit_3;
GVL.IIVD.S_Str_Pmp_Em_Run_FOC.x			:= GVL.IIVD.S_Str_Pmp_Em_Run_FOC.v AND _FB_CanRx_Message_Unpack_211.S_Bit_2;
GVL.IIVD.S_Str_Pmp_Em_Run_FOC.e			:= _FB_CanRx_Message_Unpack_211.S_Bit_3 AND NOT _FB_CanRx_Message_Unpack_211.S_Bit_2 ;
GVL.IIVD.S_Str_Pmp_Em_Run_FOC.na		:= _FB_CanRx_Message_Unpack_211.S_Bit_3 AND _FB_CanRx_Message_Unpack_211.S_Bit_2 ;
{endregion}
{region " SIGNAL AREA : NAME->S_Str_Pmp_Em_Run_Slp LENGTH->2 STARTBIT :4"}
GVL.IIVD.S_Str_Pmp_Em_Run_Slp.v			:= NOT GVL.IIVD.S_TmOut_Direksiyon_Pompasi_Durum_0X211 AND NOT _FB_CanRx_Message_Unpack_211.S_Bit_5;
GVL.IIVD.S_Str_Pmp_Em_Run_Slp.x			:= GVL.IIVD.S_Str_Pmp_Em_Run_Slp.v AND _FB_CanRx_Message_Unpack_211.S_Bit_4;
GVL.IIVD.S_Str_Pmp_Em_Run_Slp.e			:= _FB_CanRx_Message_Unpack_211.S_Bit_5 AND NOT _FB_CanRx_Message_Unpack_211.S_Bit_4 ;
GVL.IIVD.S_Str_Pmp_Em_Run_Slp.na		:= _FB_CanRx_Message_Unpack_211.S_Bit_5 AND _FB_CanRx_Message_Unpack_211.S_Bit_4 ;
{endregion}
{region " SIGNAL AREA : NAME->S_ER_Str_Pmp LENGTH->2 STARTBIT :6"}
GVL.IIVD.S_ER_Str_Pmp.v					:= NOT GVL.IIVD.S_TmOut_Direksiyon_Pompasi_Durum_0X211 AND NOT _FB_CanRx_Message_Unpack_211.S_Bit_7;
GVL.IIVD.S_ER_Str_Pmp.x					:= GVL.IIVD.S_ER_Str_Pmp.v AND _FB_CanRx_Message_Unpack_211.S_Bit_6;
GVL.IIVD.S_ER_Str_Pmp.e					:= _FB_CanRx_Message_Unpack_211.S_Bit_7 AND NOT _FB_CanRx_Message_Unpack_211.S_Bit_6 ;
GVL.IIVD.S_ER_Str_Pmp.na				:= _FB_CanRx_Message_Unpack_211.S_Bit_7 AND _FB_CanRx_Message_Unpack_211.S_Bit_6 ;
{endregion}
{region " SIGNAL AREA : NAME->S_Str_Pmp_Run LENGTH->2 STARTBIT :8"}
GVL.IIVD.S_Str_Pmp_Run.v				:= NOT GVL.IIVD.S_TmOut_Direksiyon_Pompasi_Durum_0X211 AND NOT _FB_CanRx_Message_Unpack_211.S_Bit_9;
GVL.IIVD.S_Str_Pmp_Run.x				:= GVL.IIVD.S_Str_Pmp_Run.v AND _FB_CanRx_Message_Unpack_211.S_Bit_8;
GVL.IIVD.S_Str_Pmp_Run.e				:= _FB_CanRx_Message_Unpack_211.S_Bit_9 AND NOT _FB_CanRx_Message_Unpack_211.S_Bit_8 ;
GVL.IIVD.S_Str_Pmp_Run.na				:= _FB_CanRx_Message_Unpack_211.S_Bit_9 AND _FB_CanRx_Message_Unpack_211.S_Bit_8 ;
{endregion}
{region " SIGNAL AREA : NAME->X_T_Str_Pmp_Mot LENGTH->8 STARTBIT :16"}
Raw_X_T_Str_Pmp_Mot						:= _FB_CanRx_Message_Unpack_211.X_Byte_2;
GVL.IIVD.X_T_Str_Pmp_Mot.e				:= (Raw_X_T_Str_Pmp_Mot > 16#FD) AND (Raw_X_T_Str_Pmp_Mot < 16#FF);
GVL.IIVD.X_T_Str_Pmp_Mot.na				:= (Raw_X_T_Str_Pmp_Mot = 16#FF);
GVL.IIVD.X_T_Str_Pmp_Mot.RangeExcd		:= NOT ((USINT_TO_REAL(BYTE_TO_USINT(Raw_X_T_Str_Pmp_Mot))+(-40) >= -40) AND (USINT_TO_REAL(BYTE_TO_USINT(Raw_X_T_Str_Pmp_Mot))+(-40) <= 200));
GVL.IIVD.X_T_Str_Pmp_Mot.v				:= NOT( GVL.IIVD.S_TmOut_Direksiyon_Pompasi_Durum_0X211 OR GVL.IIVD.X_T_Str_Pmp_Mot.RangeExcd OR GVL.IIVD.X_T_Str_Pmp_Mot.e OR GVL.IIVD.X_T_Str_Pmp_Mot.na) ;
GVL.IIVD.X_T_Str_Pmp_Mot.x				:= 
(*SELECT 1 : Is data valid ?*)				SEL(GVL.IIVD.X_T_Str_Pmp_Mot.v,
(*DEFAULT value assigment*)					0,
(*Transmission is VALID*)					USINT_TO_REAL(BYTE_TO_USINT(Raw_X_T_Str_Pmp_Mot))+(-40));
{endregion}
{region " SIGNAL AREA : NAME->X_T_Str_Pmp_Inver LENGTH->8 STARTBIT :24"}
Raw_X_T_Str_Pmp_Inver					:= _FB_CanRx_Message_Unpack_211.X_Byte_3;
GVL.IIVD.X_T_Str_Pmp_Inver.e			:= (Raw_X_T_Str_Pmp_Inver > 16#FD) AND (Raw_X_T_Str_Pmp_Inver < 16#FF);
GVL.IIVD.X_T_Str_Pmp_Inver.na			:= (Raw_X_T_Str_Pmp_Inver = 16#FF);
GVL.IIVD.X_T_Str_Pmp_Inver.RangeExcd	:= NOT ((USINT_TO_REAL(BYTE_TO_USINT(Raw_X_T_Str_Pmp_Inver))+(-40) >= -40) AND (USINT_TO_REAL(BYTE_TO_USINT(Raw_X_T_Str_Pmp_Inver))+(-40) <= 170));
GVL.IIVD.X_T_Str_Pmp_Inver.v			:= NOT( GVL.IIVD.S_TmOut_Direksiyon_Pompasi_Durum_0X211 OR GVL.IIVD.X_T_Str_Pmp_Inver.RangeExcd OR GVL.IIVD.X_T_Str_Pmp_Inver.e OR GVL.IIVD.X_T_Str_Pmp_Inver.na) ;
GVL.IIVD.X_T_Str_Pmp_Inver.x			:= 
(*SELECT 1 : Is data valid ?*)				SEL(GVL.IIVD.X_T_Str_Pmp_Inver.v,
(*DEFAULT value assigment*)					0,
(*Transmission is VALID*)					USINT_TO_REAL(BYTE_TO_USINT(Raw_X_T_Str_Pmp_Inver))+(-40));
{endregion}
{region " SIGNAL AREA : NAME->X_Mot_Load_Str_Pmp LENGTH->8 STARTBIT :32"}
Raw_X_Mot_Load_Str_Pmp					:= _FB_CanRx_Message_Unpack_211.X_Byte_4;
GVL.IIVD.X_Mot_Load_Str_Pmp.e			:= (Raw_X_Mot_Load_Str_Pmp > 16#FD) AND (Raw_X_Mot_Load_Str_Pmp < 16#FF);
GVL.IIVD.X_Mot_Load_Str_Pmp.na			:= (Raw_X_Mot_Load_Str_Pmp = 16#FF);
GVL.IIVD.X_Mot_Load_Str_Pmp.RangeExcd	:= NOT ((USINT_TO_REAL(BYTE_TO_USINT(Raw_X_Mot_Load_Str_Pmp)) >= -100) AND (USINT_TO_REAL(BYTE_TO_USINT(Raw_X_Mot_Load_Str_Pmp)) <= 100));
GVL.IIVD.X_Mot_Load_Str_Pmp.v			:= NOT( GVL.IIVD.S_TmOut_Direksiyon_Pompasi_Durum_0X211 OR GVL.IIVD.X_Mot_Load_Str_Pmp.RangeExcd OR GVL.IIVD.X_Mot_Load_Str_Pmp.e OR GVL.IIVD.X_Mot_Load_Str_Pmp.na) ;
GVL.IIVD.X_Mot_Load_Str_Pmp.x			:= 
(*SELECT 1 : Is data valid ?*)				SEL(GVL.IIVD.X_Mot_Load_Str_Pmp.v,
(*DEFAULT value assigment*)					0,
(*Transmission is VALID*)					USINT_TO_REAL(BYTE_TO_USINT(Raw_X_Mot_Load_Str_Pmp)));
{endregion}
{region " SIGNAL AREA : NAME->X_T_Air_Cmp LENGTH->8 STARTBIT :48"}
Raw_X_T_Air_Cmp							:= _FB_CanRx_Message_Unpack_211.X_Byte_6;
GVL.IIVD.X_T_Air_Cmp.e					:= (Raw_X_T_Air_Cmp > 16#FD) AND (Raw_X_T_Air_Cmp < 16#FF);
GVL.IIVD.X_T_Air_Cmp.na					:= (Raw_X_T_Air_Cmp = 16#FF);
GVL.IIVD.X_T_Air_Cmp.RangeExcd			:= NOT ((USINT_TO_REAL(BYTE_TO_USINT(Raw_X_T_Air_Cmp))+(-40) >= -40) AND (USINT_TO_REAL(BYTE_TO_USINT(Raw_X_T_Air_Cmp))+(-40) <= 215));
GVL.IIVD.X_T_Air_Cmp.v					:= NOT( GVL.IIVD.S_TmOut_Direksiyon_Pompasi_Durum_0X211 OR GVL.IIVD.X_T_Air_Cmp.RangeExcd OR GVL.IIVD.X_T_Air_Cmp.e OR GVL.IIVD.X_T_Air_Cmp.na) ;
GVL.IIVD.X_T_Air_Cmp.x					:= 
(*SELECT 1 : Is data valid ?*)				SEL(GVL.IIVD.X_T_Air_Cmp.v,
(*DEFAULT value assigment*)					0,
(*Transmission is VALID*)					USINT_TO_REAL(BYTE_TO_USINT(Raw_X_T_Air_Cmp))+(-40));
{endregion}		  
{region " SIGNAL AREA : NAME->S_ER_Air_Cmp_Tmp LENGTH->2 STARTBIT :56"}
GVL.IIVD.S_ER_Air_Cmp_Tmp.v				:= NOT GVL.IIVD.S_TmOut_Direksiyon_Pompasi_Durum_0X211 AND NOT _FB_CanRx_Message_Unpack_211.S_Bit_57;
GVL.IIVD.S_ER_Air_Cmp_Tmp.x				:= GVL.IIVD.S_ER_Air_Cmp_Tmp.v AND _FB_CanRx_Message_Unpack_211.S_Bit_56;
GVL.IIVD.S_ER_Air_Cmp_Tmp.e				:= _FB_CanRx_Message_Unpack_211.S_Bit_57 AND NOT _FB_CanRx_Message_Unpack_211.S_Bit_56 ;
GVL.IIVD.S_ER_Air_Cmp_Tmp.na			:= _FB_CanRx_Message_Unpack_211.S_Bit_57 AND _FB_CanRx_Message_Unpack_211.S_Bit_56 ;
{endregion}
{region " SIGNAL AREA : NAME->S_Air_Cmp_Filt_Warn_Actv LENGTH->2 STARBIT :58"}
GVL.IIVD.S_Air_Cmp_Filt_Warn_Actv.v		:= NOT GVL.IIVD.S_TmOut_Direksiyon_Pompasi_Durum_0X211 AND NOT _FB_CanRx_Message_Unpack_211.S_Bit_59;
GVL.IIVD.S_Air_Cmp_Filt_Warn_Actv.x		:= GVL.IIVD.S_Air_Cmp_Filt_Warn_Actv.v AND _FB_CanRx_Message_Unpack_211.S_Bit_58;
GVL.IIVD.S_Air_Cmp_Filt_Warn_Actv.e		:= _FB_CanRx_Message_Unpack_211.S_Bit_59 AND NOT _FB_CanRx_Message_Unpack_211.S_Bit_58;
GVL.IIVD.S_Air_Cmp_Filt_Warn_Actv.na	:= _FB_CanRx_Message_Unpack_211.S_Bit_59 AND _FB_CanRx_Message_Unpack_211.S_Bit_58;
{endregion}
{endregion}

{region " MESSAGE AREA :Arac_Durumlari- ID:220"}

_FB_CanRx_Message_Unpack_220 (	C_Enable	:= GVL.IIVD.S_CAN_Init,
     							Obj_CAN		:= ADR(GVL.IC.Obj_CAN0),
     							X_MsgID		:= 16#220,
     							Tm_MsgTmOut	:= TIME#2500MS,
     							S_Extended	:= 0,
     							S_ER_TmOut	=> GVL.IIVD.S_TmOut_Arac_Durumlari_0X220);

{region " SIGNAL AREA : NAME->S_Hld_Brk_Byp LENGTH->2 STARTBIT :0"}
GVL.IIVD.S_Hld_Brk_Byp.v				:= NOT GVL.IIVD.S_TmOut_Arac_Durumlari_0X220 AND NOT _FB_CanRx_Message_Unpack_220.S_Bit_1;
GVL.IIVD.S_Hld_Brk_Byp.x				:= GVL.IIVD.S_Hld_Brk_Byp.v AND _FB_CanRx_Message_Unpack_220.S_Bit_0;
GVL.IIVD.S_Hld_Brk_Byp.e				:= _FB_CanRx_Message_Unpack_220.S_Bit_1 AND NOT _FB_CanRx_Message_Unpack_220.S_Bit_0 ;
GVL.IIVD.S_Hld_Brk_Byp.na				:= _FB_CanRx_Message_Unpack_220.S_Bit_1 AND _FB_CanRx_Message_Unpack_220.S_Bit_0 ;
{endregion}
{region " SIGNAL AREA : NAME->S_Hld_Brk_Req LENGTH->2 STARTBIT :2"}
GVL.IIVD.S_Hld_Brk_Req.v				:= NOT GVL.IIVD.S_TmOut_Arac_Durumlari_0X220 AND NOT _FB_CanRx_Message_Unpack_220.S_Bit_3;
GVL.IIVD.S_Hld_Brk_Req.x				:= GVL.IIVD.S_Hld_Brk_Req.v AND _FB_CanRx_Message_Unpack_220.S_Bit_2;
GVL.IIVD.S_Hld_Brk_Req.e				:= _FB_CanRx_Message_Unpack_220.S_Bit_3 AND NOT _FB_CanRx_Message_Unpack_220.S_Bit_2 ;
GVL.IIVD.S_Hld_Brk_Req.na				:= _FB_CanRx_Message_Unpack_220.S_Bit_3 AND _FB_CanRx_Message_Unpack_220.S_Bit_2 ;
{endregion}
{region " SIGNAL AREA : NAME->S_Hld_Brk_Actv LENGTH->2 STARTBIT :4"}
GVL.IIVD.S_Hld_Brk_Actv.v				:= NOT GVL.IIVD.S_TmOut_Arac_Durumlari_0X220 AND NOT _FB_CanRx_Message_Unpack_220.S_Bit_5;
GVL.IIVD.S_Hld_Brk_Actv.x				:= GVL.IIVD.S_Hld_Brk_Actv.v AND _FB_CanRx_Message_Unpack_220.S_Bit_4;
GVL.IIVD.S_Hld_Brk_Actv.e				:= _FB_CanRx_Message_Unpack_220.S_Bit_5 AND NOT _FB_CanRx_Message_Unpack_220.S_Bit_4 ;
GVL.IIVD.S_Hld_Brk_Actv.na				:= _FB_CanRx_Message_Unpack_220.S_Bit_5 AND _FB_CanRx_Message_Unpack_220.S_Bit_4 ;
{endregion}
{region " SIGNAL AREA : NAME->S_Aut_Lub_Oil_Lv_Lo LENGTH->2 STARTBIT :6"}
GVL.IIVD.S_Aut_Lub_Oil_Lv_Lo.v			:= NOT GVL.IIVD.S_TmOut_Arac_Durumlari_0X220 AND NOT _FB_CanRx_Message_Unpack_220.S_Bit_7;
GVL.IIVD.S_Aut_Lub_Oil_Lv_Lo.x			:= GVL.IIVD.S_Aut_Lub_Oil_Lv_Lo.v AND _FB_CanRx_Message_Unpack_220.S_Bit_6;
GVL.IIVD.S_Aut_Lub_Oil_Lv_Lo.e			:= _FB_CanRx_Message_Unpack_220.S_Bit_7 AND NOT _FB_CanRx_Message_Unpack_220.S_Bit_6 ;
GVL.IIVD.S_Aut_Lub_Oil_Lv_Lo.na			:= _FB_CanRx_Message_Unpack_220.S_Bit_7 AND _FB_CanRx_Message_Unpack_220.S_Bit_6 ;
{endregion}
{region " SIGNAL AREA : NAME->S_ECAS_Dwn_Req LENGTH->2 STARTBIT :8"}
GVL.IIVD.S_ECAS_Dwn_Req.v				:= NOT GVL.IIVD.S_TmOut_Arac_Durumlari_0X220 AND NOT _FB_CanRx_Message_Unpack_220.S_Bit_9;
GVL.IIVD.S_ECAS_Dwn_Req.x				:= GVL.IIVD.S_ECAS_Dwn_Req.v AND _FB_CanRx_Message_Unpack_220.S_Bit_8;
GVL.IIVD.S_ECAS_Dwn_Req.e				:= _FB_CanRx_Message_Unpack_220.S_Bit_9 AND NOT _FB_CanRx_Message_Unpack_220.S_Bit_8 ;
GVL.IIVD.S_ECAS_Dwn_Req.na				:= _FB_CanRx_Message_Unpack_220.S_Bit_9 AND _FB_CanRx_Message_Unpack_220.S_Bit_8 ;
{endregion}
{region " SIGNAL AREA : NAME->S_ECAS_Up_Req LENGTH->2 STARTBIT :10"}
GVL.IIVD.S_ECAS_Up_Req.v				:= NOT GVL.IIVD.S_TmOut_Arac_Durumlari_0X220 AND NOT _FB_CanRx_Message_Unpack_220.S_Bit_11;
GVL.IIVD.S_ECAS_Up_Req.x				:= GVL.IIVD.S_ECAS_Up_Req.v AND _FB_CanRx_Message_Unpack_220.S_Bit_10;
GVL.IIVD.S_ECAS_Up_Req.e				:= _FB_CanRx_Message_Unpack_220.S_Bit_11 AND NOT _FB_CanRx_Message_Unpack_220.S_Bit_10 ;
GVL.IIVD.S_ECAS_Up_Req.na				:= _FB_CanRx_Message_Unpack_220.S_Bit_11 AND _FB_CanRx_Message_Unpack_220.S_Bit_10 ;
{endregion}
{region " SIGNAL AREA : NAME->S_ECAS_Pos_Down LENGTH->2 STARTBIT :12"}
GVL.IIVD.S_ECAS_Pos_Down.v				:= NOT GVL.IIVD.S_TmOut_Arac_Durumlari_0X220 AND NOT _FB_CanRx_Message_Unpack_220.S_Bit_13;
GVL.IIVD.S_ECAS_Pos_Down.x				:= GVL.IIVD.S_ECAS_Pos_Down.v AND _FB_CanRx_Message_Unpack_220.S_Bit_12;
GVL.IIVD.S_ECAS_Pos_Down.e				:= _FB_CanRx_Message_Unpack_220.S_Bit_13 AND NOT _FB_CanRx_Message_Unpack_220.S_Bit_12 ;
GVL.IIVD.S_ECAS_Pos_Down.na				:= _FB_CanRx_Message_Unpack_220.S_Bit_13 AND _FB_CanRx_Message_Unpack_220.S_Bit_12 ;
{endregion}
{region " SIGNAL AREA : NAME->S_ECAS_Pos_Up LENGTH->2 STARTBIT :14"}
GVL.IIVD.S_ECAS_Pos_Up.v				:= NOT GVL.IIVD.S_TmOut_Arac_Durumlari_0X220 AND NOT _FB_CanRx_Message_Unpack_220.S_Bit_15;
GVL.IIVD.S_ECAS_Pos_Up.x				:= GVL.IIVD.S_ECAS_Pos_Up.v AND _FB_CanRx_Message_Unpack_220.S_Bit_14;
GVL.IIVD.S_ECAS_Pos_Up.e				:= _FB_CanRx_Message_Unpack_220.S_Bit_15 AND NOT _FB_CanRx_Message_Unpack_220.S_Bit_14 ;
GVL.IIVD.S_ECAS_Pos_Up.na				:= _FB_CanRx_Message_Unpack_220.S_Bit_15 AND _FB_CanRx_Message_Unpack_220.S_Bit_14 ;
{endregion}
{region " SIGNAL AREA : NAME->S_Knl_Req LENGTH->2 STARTBIT :16"}
GVL.IIVD.S_Knl_Req.v					:= NOT GVL.IIVD.S_TmOut_Arac_Durumlari_0X220 AND NOT _FB_CanRx_Message_Unpack_220.S_Bit_17;
GVL.IIVD.S_Knl_Req.x					:= GVL.IIVD.S_Knl_Req.v AND _FB_CanRx_Message_Unpack_220.S_Bit_16;
GVL.IIVD.S_Knl_Req.e					:= _FB_CanRx_Message_Unpack_220.S_Bit_17 AND NOT _FB_CanRx_Message_Unpack_220.S_Bit_16 ;
GVL.IIVD.S_Knl_Req.na					:= _FB_CanRx_Message_Unpack_220.S_Bit_17 AND _FB_CanRx_Message_Unpack_220.S_Bit_16 ;
{endregion}
{region " SIGNAL AREA : NAME->S_Knl_Actv LENGTH->2 STARTBIT :18"}
GVL.IIVD.S_Knl_Actv.v					:= NOT GVL.IIVD.S_TmOut_Arac_Durumlari_0X220 AND NOT _FB_CanRx_Message_Unpack_220.S_Bit_19;
GVL.IIVD.S_Knl_Actv.x					:= GVL.IIVD.S_Knl_Actv.v AND _FB_CanRx_Message_Unpack_220.S_Bit_18;
GVL.IIVD.S_Knl_Actv.e					:= _FB_CanRx_Message_Unpack_220.S_Bit_19 AND NOT _FB_CanRx_Message_Unpack_220.S_Bit_18 ;
GVL.IIVD.S_Knl_Actv.na					:= _FB_CanRx_Message_Unpack_220.S_Bit_19 AND _FB_CanRx_Message_Unpack_220.S_Bit_18 ;
{endregion}
{region " SIGNAL AREA : NAME->S_Fwd_Gear LENGTH->2 STARTBIT :20"}
GVL.IIVD.S_Fwd_Gear.v					:= NOT GVL.IIVD.S_TmOut_Arac_Durumlari_0X220 AND NOT _FB_CanRx_Message_Unpack_220.S_Bit_21;
GVL.IIVD.S_Fwd_Gear.x					:= GVL.IIVD.S_Fwd_Gear.v AND _FB_CanRx_Message_Unpack_220.S_Bit_20;
GVL.IIVD.S_Fwd_Gear.e					:= _FB_CanRx_Message_Unpack_220.S_Bit_21 AND NOT _FB_CanRx_Message_Unpack_220.S_Bit_20 ;
GVL.IIVD.S_Fwd_Gear.na					:= _FB_CanRx_Message_Unpack_220.S_Bit_21 AND _FB_CanRx_Message_Unpack_220.S_Bit_20 ;
{endregion}
{region " SIGNAL AREA : NAME->S_Bwd_Gear LENGTH->2 STARTBIT :22"}
GVL.IIVD.S_Bwd_Gear.v					:= NOT GVL.IIVD.S_TmOut_Arac_Durumlari_0X220 AND NOT _FB_CanRx_Message_Unpack_220.S_Bit_23;
GVL.IIVD.S_Bwd_Gear.x					:= GVL.IIVD.S_Bwd_Gear.v AND _FB_CanRx_Message_Unpack_220.S_Bit_22;
GVL.IIVD.S_Bwd_Gear.e					:= _FB_CanRx_Message_Unpack_220.S_Bit_23 AND NOT _FB_CanRx_Message_Unpack_220.S_Bit_22 ;
GVL.IIVD.S_Bwd_Gear.na					:= _FB_CanRx_Message_Unpack_220.S_Bit_23 AND _FB_CanRx_Message_Unpack_220.S_Bit_22 ;
{endregion}
{region " SIGNAL AREA : NAME->S_Vh_Actv_Key_Lv1 LENGTH->2 STARTBIT :24"}
GVL.IIVD.S_Vh_Actv_Key_Lv1.v			:= NOT GVL.IIVD.S_TmOut_Arac_Durumlari_0X220 AND NOT _FB_CanRx_Message_Unpack_220.S_Bit_25;
GVL.IIVD.S_Vh_Actv_Key_Lv1.x			:= GVL.IIVD.S_Vh_Actv_Key_Lv1.v AND _FB_CanRx_Message_Unpack_220.S_Bit_24;
GVL.IIVD.S_Vh_Actv_Key_Lv1.e			:= _FB_CanRx_Message_Unpack_220.S_Bit_25 AND NOT _FB_CanRx_Message_Unpack_220.S_Bit_24 ;
GVL.IIVD.S_Vh_Actv_Key_Lv1.na			:= _FB_CanRx_Message_Unpack_220.S_Bit_25 AND _FB_CanRx_Message_Unpack_220.S_Bit_24 ;
{endregion}
{region " SIGNAL AREA : NAME->S_Vh_Actv_Key_Lv2 LENGTH->2 STARTBIT :26"}
GVL.IIVD.S_Vh_Actv_Key_Lv2.v			:= NOT GVL.IIVD.S_TmOut_Arac_Durumlari_0X220 AND NOT _FB_CanRx_Message_Unpack_220.S_Bit_27;
GVL.IIVD.S_Vh_Actv_Key_Lv2.x			:= GVL.IIVD.S_Vh_Actv_Key_Lv2.v AND _FB_CanRx_Message_Unpack_220.S_Bit_26;
GVL.IIVD.S_Vh_Actv_Key_Lv2.e			:= _FB_CanRx_Message_Unpack_220.S_Bit_27 AND NOT _FB_CanRx_Message_Unpack_220.S_Bit_26 ;
GVL.IIVD.S_Vh_Actv_Key_Lv2.na			:= _FB_CanRx_Message_Unpack_220.S_Bit_27 AND _FB_CanRx_Message_Unpack_220.S_Bit_26 ;
{endregion}
{region " SIGNAL AREA : NAME->S_Vh_Actv_Key_Lv3 LENGTH->2 STARTBIT :28"}
GVL.IIVD.S_Vh_Actv_Key_Lv3.v			:= NOT GVL.IIVD.S_TmOut_Arac_Durumlari_0X220 AND NOT _FB_CanRx_Message_Unpack_220.S_Bit_29;
GVL.IIVD.S_Vh_Actv_Key_Lv3.x			:= GVL.IIVD.S_Vh_Actv_Key_Lv3.v AND _FB_CanRx_Message_Unpack_220.S_Bit_28;
GVL.IIVD.S_Vh_Actv_Key_Lv3.e			:= _FB_CanRx_Message_Unpack_220.S_Bit_29 AND NOT _FB_CanRx_Message_Unpack_220.S_Bit_28 ;
GVL.IIVD.S_Vh_Actv_Key_Lv3.na			:= _FB_CanRx_Message_Unpack_220.S_Bit_29 AND _FB_CanRx_Message_Unpack_220.S_Bit_28 ;
{endregion}
{region " SIGNAL AREA : NAME->S_Brk_Park LENGTH->2 STARTBIT :30"}
GVL.IIVD.S_Brk_Park.v					:= NOT GVL.IIVD.S_TmOut_Arac_Durumlari_0X220 AND NOT _FB_CanRx_Message_Unpack_220.S_Bit_31;
GVL.IIVD.S_Brk_Park.x					:= GVL.IIVD.S_Brk_Park.v AND _FB_CanRx_Message_Unpack_220.S_Bit_30;
GVL.IIVD.S_Brk_Park.e					:= _FB_CanRx_Message_Unpack_220.S_Bit_31 AND NOT _FB_CanRx_Message_Unpack_220.S_Bit_30 ;
GVL.IIVD.S_Brk_Park.na					:= _FB_CanRx_Message_Unpack_220.S_Bit_31 AND _FB_CanRx_Message_Unpack_220.S_Bit_30 ;
{endregion}
{region " SIGNAL AREA : NAME->Z_Ret_Lv LENGTH->4 STARTBIT :32"}
_FB_PACK_8BITS_TO_BYTE_8	(	S_BIT_0		:= _FB_CanRx_Message_Unpack_220.S_Bit_32, 
								S_BIT_1		:= _FB_CanRx_Message_Unpack_220.S_Bit_33, 
								S_BIT_2		:= _FB_CanRx_Message_Unpack_220.S_Bit_34, 
								S_BIT_3		:= _FB_CanRx_Message_Unpack_220.S_Bit_35, 
								X_BYTE_0	=> Raw_Z_Ret_Lv);
GVL.IIVD.Z_Ret_Lv.e						:= (Raw_Z_Ret_Lv > 6) AND (Raw_Z_Config_Clu < 15);
GVL.IIVD.Z_Ret_Lv.na					:= (Raw_Z_Ret_Lv = 15);
GVL.IIVD.Z_Ret_Lv.RangeExcd				:= NOT (Raw_Z_Ret_Lv >= 0) AND (Raw_Z_Ret_Lv <= 15);
GVL.IIVD.Z_Ret_Lv.v						:= NOT( GVL.IIVD.S_TmOut_Arac_Durumlari_0X220 OR GVL.IIVD.Z_Ret_Lv.RangeExcd OR GVL.IIVD.Z_Ret_Lv.e OR GVL.IIVD.Z_Ret_Lv.na) ;
GVL.IIVD.Z_Ret_Lv.x						:= 
(*SELECT 1 : Is data valid ?*)				SEL(GVL.IIVD.Z_Ret_Lv.v,
(*DEFAULT value assigment*)					0,
(*Transmission is VALID*)					Raw_Z_Ret_Lv);
{endregion}	
// PR1006_SRS_000670_TIMTRO
{region " SIGNAL AREA : NAME->S_ER_Aut_Lub_Snsr LENGTH->2 STARTBIT :36"}
GVL.IIVD.S_Aut_Lub_Actv.v			:= NOT GVL.IIVD.S_TmOut_Arac_Durumlari_0X220 AND NOT _FB_CanRx_Message_Unpack_220.S_Bit_37;
GVL.IIVD.S_Aut_Lub_Actv.x			:= GVL.IIVD.S_Aut_Lub_Actv.v AND _FB_CanRx_Message_Unpack_220.S_Bit_36;
GVL.IIVD.S_Aut_Lub_Actv.e			:= _FB_CanRx_Message_Unpack_220.S_Bit_37 AND NOT _FB_CanRx_Message_Unpack_220.S_Bit_36;
GVL.IIVD.S_Aut_Lub_Actv.na			:= _FB_CanRx_Message_Unpack_220.S_Bit_37 AND _FB_CanRx_Message_Unpack_220.S_Bit_36;
{endregion}
// PR1006_SRS_000673_TIMTRO
{region " SIGNAL AREA : NAME->S_ER_Aut_Lub_Snsr LENGTH->2 STARTBIT :38"}
GVL.IIVD.S_ER_Aut_Lub_Snsr.v		:= NOT GVL.IIVD.S_TmOut_Arac_Durumlari_0X220 AND NOT _FB_CanRx_Message_Unpack_220.S_Bit_39;
GVL.IIVD.S_ER_Aut_Lub_Snsr.x		:= GVL.IIVD.S_ER_Aut_Lub_Snsr.v AND _FB_CanRx_Message_Unpack_220.S_Bit_38;
GVL.IIVD.S_ER_Aut_Lub_Snsr.e		:= _FB_CanRx_Message_Unpack_220.S_Bit_39 AND NOT _FB_CanRx_Message_Unpack_220.S_Bit_38;
GVL.IIVD.S_ER_Aut_Lub_Snsr.na		:= _FB_CanRx_Message_Unpack_220.S_Bit_39 AND _FB_CanRx_Message_Unpack_220.S_Bit_38;
{endregion}
{region " SIGNAL AREA : NAME->S_Bat_Mod_Btn LENGTH->2 STARTBIT :42"}
GVL.IIVD.S_Bat_Mod_Btn.v				:= NOT GVL.IIVD.S_TmOut_Arac_Durumlari_0X220 AND NOT _FB_CanRx_Message_Unpack_220.S_Bit_43;
GVL.IIVD.S_Bat_Mod_Btn.x				:= GVL.IIVD.S_Bat_Mod_Btn.v AND _FB_CanRx_Message_Unpack_220.S_Bit_42;
GVL.IIVD.S_Bat_Mod_Btn.e				:= _FB_CanRx_Message_Unpack_220.S_Bit_43 AND NOT _FB_CanRx_Message_Unpack_220.S_Bit_42 ;
GVL.IIVD.S_Bat_Mod_Btn.na				:= _FB_CanRx_Message_Unpack_220.S_Bit_43 AND _FB_CanRx_Message_Unpack_220.S_Bit_42 ;
{endregion}		  
{region " SIGNAL AREA : NAME->S_Bat_Mod_Btn LENGTH->2 STARTBIT :44"}
GVL.IIVD.S_Elec_Mod_Btn.v				:= NOT GVL.IIVD.S_TmOut_Arac_Durumlari_0X220 AND NOT _FB_CanRx_Message_Unpack_220.S_Bit_45;
GVL.IIVD.S_Elec_Mod_Btn.x				:= GVL.IIVD.S_Elec_Mod_Btn.v AND _FB_CanRx_Message_Unpack_220.S_Bit_44;
GVL.IIVD.S_Elec_Mod_Btn.e				:= _FB_CanRx_Message_Unpack_220.S_Bit_45 AND NOT _FB_CanRx_Message_Unpack_220.S_Bit_44 ;
GVL.IIVD.S_Elec_Mod_Btn.na				:= _FB_CanRx_Message_Unpack_220.S_Bit_45 AND _FB_CanRx_Message_Unpack_220.S_Bit_44 ;
{endregion}
{region " SIGNAL AREA : NAME->S_Bwd_Lft_Chrg_Btn LENGTH->2 STARTBIT :46"}
GVL.IIVD.S_Bwd_Lft_Chrg_Btn.v				:= NOT GVL.IIVD.S_TmOut_Arac_Durumlari_0X220 AND NOT _FB_CanRx_Message_Unpack_220.S_Bit_47;
GVL.IIVD.S_Bwd_Lft_Chrg_Btn.x				:= GVL.IIVD.S_Bwd_Lft_Chrg_Btn.v AND _FB_CanRx_Message_Unpack_220.S_Bit_46;
GVL.IIVD.S_Bwd_Lft_Chrg_Btn.e				:= _FB_CanRx_Message_Unpack_220.S_Bit_47 AND NOT _FB_CanRx_Message_Unpack_220.S_Bit_46;
GVL.IIVD.S_Bwd_Lft_Chrg_Btn.na				:= _FB_CanRx_Message_Unpack_220.S_Bit_47 AND _FB_CanRx_Message_Unpack_220.S_Bit_46;
{endregion}
{region " SIGNAL AREA : NAME->S_Bwd_Lft_Chrg_Em_Stop_Swc1 LENGTH->2 STARTBIT :48"}
GVL.IIVD.S_Bwd_Lft_Chrg_Em_Stop_Swc1.v		:= NOT GVL.IIVD.S_TmOut_Arac_Durumlari_0X220 AND NOT _FB_CanRx_Message_Unpack_220.S_Bit_49;
GVL.IIVD.S_Bwd_Lft_Chrg_Em_Stop_Swc1.x		:= GVL.IIVD.S_Bwd_Lft_Chrg_Em_Stop_Swc1.v AND _FB_CanRx_Message_Unpack_220.S_Bit_48;
GVL.IIVD.S_Bwd_Lft_Chrg_Em_Stop_Swc1.e		:= _FB_CanRx_Message_Unpack_220.S_Bit_49 AND NOT _FB_CanRx_Message_Unpack_220.S_Bit_48;
GVL.IIVD.S_Bwd_Lft_Chrg_Em_Stop_Swc1.na		:= _FB_CanRx_Message_Unpack_220.S_Bit_49 AND _FB_CanRx_Message_Unpack_220.S_Bit_48;
{endregion}
{region " SIGNAL AREA : NAME->S_Bwd_Lft_Chrg_Em_Stop_Swc2 LENGTH->2 STARTBIT :50"}
GVL.IIVD.S_Bwd_Lft_Chrg_Em_Stop_Swc2.v		:= NOT GVL.IIVD.S_TmOut_Arac_Durumlari_0X220 AND NOT _FB_CanRx_Message_Unpack_220.S_Bit_51;
GVL.IIVD.S_Bwd_Lft_Chrg_Em_Stop_Swc2.x		:= GVL.IIVD.S_Bwd_Lft_Chrg_Em_Stop_Swc2.v AND _FB_CanRx_Message_Unpack_220.S_Bit_50;
GVL.IIVD.S_Bwd_Lft_Chrg_Em_Stop_Swc2.e		:= _FB_CanRx_Message_Unpack_220.S_Bit_51 AND NOT _FB_CanRx_Message_Unpack_220.S_Bit_50;
GVL.IIVD.S_Bwd_Lft_Chrg_Em_Stop_Swc2.na		:= _FB_CanRx_Message_Unpack_220.S_Bit_51 AND _FB_CanRx_Message_Unpack_220.S_Bit_50;
{endregion}
{region " SIGNAL AREA : NAME->Z_Config_Clu LENGTH->8 STARTBIT :56"}
Raw_Z_Config_Clu						:= _FB_CanRx_Message_Unpack_220.X_Byte_7;
GVL.IIVD.Z_Config_Clu.e					:= (Raw_Z_Config_Clu > 16#FD) AND (Raw_Z_Config_Clu < 16#FF);
GVL.IIVD.Z_Config_Clu.na				:= (Raw_Z_Config_Clu = 16#FF);
GVL.IIVD.Z_Config_Clu.RangeExcd			:= NOT (Raw_Z_Config_Clu >= 0) AND (Raw_Z_Config_Clu <= 15);
GVL.IIVD.Z_Config_Clu.v					:= NOT( GVL.IIVD.S_TmOut_Arac_Durumlari_0X220 OR GVL.IIVD.Z_Config_Clu.RangeExcd OR GVL.IIVD.Z_Config_Clu.e OR GVL.IIVD.Z_Config_Clu.na) ;
GVL.IIVD.Z_Config_Clu.x					:= 
(*SELECT 1 : Is data valid ?*)				SEL(GVL.IIVD.Z_Config_Clu.v,
(*DEFAULT value assigment*)					0,
(*Transmission is VALID*)					Raw_Z_Config_Clu);
{endregion}		  
{endregion}
{region " MESSAGE AREA :Fren_balata_durumlari- ID:221"}

_FB_CanRx_Message_221 (		C_Enable	:= GVL.IIVD.S_CAN_Init,
     						Obj_CAN		:= ADR(GVL.IC.Obj_CAN0),
     						X_MsgID		:= 16#221,
     						Tm_MsgTmOut	:= TIME#2500MS,
     						S_Extended	:= 0,
     						S_ER_TmOut	=> GVL.IIVD.S_TmOut_Fren_balata_durumlari_0X221);

{region " SIGNAL AREA : NAME->X_Axl1_Brk_Ling_1 LENGTH->8 STARTBIT :0"}
Raw_X_Axl1_Brk_Ling_1					:= _FB_CanRx_Message_221.X_Byte_0;
GVL.IIVD.X_Axl1_Brk_Ling_1.e			:= (Raw_X_Axl1_Brk_Ling_1 > 16#FD) AND (Raw_X_Axl1_Brk_Ling_1 < 16#FF);
GVL.IIVD.X_Axl1_Brk_Ling_1.na			:= (Raw_X_Axl1_Brk_Ling_1 = 16#FF);
GVL.IIVD.X_Axl1_Brk_Ling_1.RangeExcd	:= NOT ((USINT_TO_REAL(BYTE_TO_USINT(Raw_X_Axl1_Brk_Ling_1)) >= 0) AND (USINT_TO_REAL(BYTE_TO_USINT(Raw_X_Axl1_Brk_Ling_1)) <= 100));
GVL.IIVD.X_Axl1_Brk_Ling_1.v			:= NOT( GVL.IIVD.S_TmOut_Fren_balata_durumlari_0X221 OR GVL.IIVD.X_Axl1_Brk_Ling_1.RangeExcd OR GVL.IIVD.X_Axl1_Brk_Ling_1.e OR GVL.IIVD.X_Axl1_Brk_Ling_1.na) ;
GVL.IIVD.X_Axl1_Brk_Ling_1.x			:= 
(*SELECT 1 : Is data valid ?*)				SEL(GVL.IIVD.X_Axl1_Brk_Ling_1.v,
(*DEFAULT value assigment*)					0,
(*Transmission is VALID*)					USINT_TO_REAL(BYTE_TO_USINT(Raw_X_Axl1_Brk_Ling_1)));
{endregion}
{region " SIGNAL AREA : NAME->X_Axl1_Brk_Ling_2 LENGTH->8 STARTBIT :8"}
Raw_X_Axl1_Brk_Ling_2					:= _FB_CanRx_Message_221.X_Byte_1;
GVL.IIVD.X_Axl1_Brk_Ling_2.e			:= (Raw_X_Axl1_Brk_Ling_2 > 16#FD) AND (Raw_X_Axl1_Brk_Ling_2 < 16#FF);
GVL.IIVD.X_Axl1_Brk_Ling_2.na			:= (Raw_X_Axl1_Brk_Ling_2 = 16#FF);
GVL.IIVD.X_Axl1_Brk_Ling_2.RangeExcd	:= NOT ((USINT_TO_REAL(BYTE_TO_USINT(Raw_X_Axl1_Brk_Ling_2)) >= 0) AND (USINT_TO_REAL(BYTE_TO_USINT(Raw_X_Axl1_Brk_Ling_2)) <= 100));
GVL.IIVD.X_Axl1_Brk_Ling_2.v			:= NOT( GVL.IIVD.S_TmOut_Fren_balata_durumlari_0X221 OR GVL.IIVD.X_Axl1_Brk_Ling_2.RangeExcd OR GVL.IIVD.X_Axl1_Brk_Ling_2.e OR GVL.IIVD.X_Axl1_Brk_Ling_2.na) ;
GVL.IIVD.X_Axl1_Brk_Ling_2.x			:= 
(*SELECT 1 : Is data valid ?*)				SEL(GVL.IIVD.X_Axl1_Brk_Ling_2.v,
(*DEFAULT value assigment*)					0,
(*Transmission is VALID*)					USINT_TO_REAL(BYTE_TO_USINT(Raw_X_Axl1_Brk_Ling_2)));
{endregion}
{region " SIGNAL AREA : NAME->X_Axl2_Brk_Ling_1 LENGTH->8 STARTBIT :16"}
Raw_X_Axl2_Brk_Ling_1					:= _FB_CanRx_Message_221.X_Byte_2;
GVL.IIVD.X_Axl2_Brk_Ling_1.e			:= (Raw_X_Axl2_Brk_Ling_1 > 16#FD) AND (Raw_X_Axl2_Brk_Ling_1 < 16#FF);
GVL.IIVD.X_Axl2_Brk_Ling_1.na			:= (Raw_X_Axl2_Brk_Ling_1 = 16#FF);
GVL.IIVD.X_Axl2_Brk_Ling_1.RangeExcd	:= NOT ((USINT_TO_REAL(BYTE_TO_USINT(Raw_X_Axl2_Brk_Ling_1)) >= 0) AND (USINT_TO_REAL(BYTE_TO_USINT(Raw_X_Axl2_Brk_Ling_1)) <= 100));
GVL.IIVD.X_Axl2_Brk_Ling_1.v			:= NOT( GVL.IIVD.S_TmOut_Fren_balata_durumlari_0X221 OR GVL.IIVD.X_Axl2_Brk_Ling_1.RangeExcd OR GVL.IIVD.X_Axl2_Brk_Ling_1.e OR GVL.IIVD.X_Axl2_Brk_Ling_1.na) ;
GVL.IIVD.X_Axl2_Brk_Ling_1.x			:= 
(*SELECT 1 : Is data valid ?*)				SEL(GVL.IIVD.X_Axl2_Brk_Ling_1.v,
(*DEFAULT value assigment*)					0,
(*Transmission is VALID*)					USINT_TO_REAL(BYTE_TO_USINT(Raw_X_Axl2_Brk_Ling_1)));
{endregion}
{region " SIGNAL AREA : NAME->X_Axl2_Brk_Ling_2 LENGTH->8 STARTBIT :24"}
Raw_X_Axl2_Brk_Ling_2					:= _FB_CanRx_Message_221.X_Byte_3;
GVL.IIVD.X_Axl2_Brk_Ling_2.e			:= (Raw_X_Axl2_Brk_Ling_2 > 16#FD) AND (Raw_X_Axl2_Brk_Ling_2 < 16#FF);
GVL.IIVD.X_Axl2_Brk_Ling_2.na			:= (Raw_X_Axl2_Brk_Ling_2 = 16#FF);
GVL.IIVD.X_Axl2_Brk_Ling_2.RangeExcd	:= NOT ((USINT_TO_REAL(BYTE_TO_USINT(Raw_X_Axl2_Brk_Ling_2)) >= 0) AND (USINT_TO_REAL(BYTE_TO_USINT(Raw_X_Axl2_Brk_Ling_2)) <= 100));
GVL.IIVD.X_Axl2_Brk_Ling_2.v			:= NOT( GVL.IIVD.S_TmOut_Fren_balata_durumlari_0X221 OR GVL.IIVD.X_Axl2_Brk_Ling_2.RangeExcd OR GVL.IIVD.X_Axl2_Brk_Ling_2.e OR GVL.IIVD.X_Axl2_Brk_Ling_2.na) ;
GVL.IIVD.X_Axl2_Brk_Ling_2.x			:= 
(*SELECT 1 : Is data valid ?*)				SEL(GVL.IIVD.X_Axl2_Brk_Ling_2.v,
(*DEFAULT value assigment*)					0,
(*Transmission is VALID*)					USINT_TO_REAL(BYTE_TO_USINT(Raw_X_Axl2_Brk_Ling_2)));
{endregion}
{region " SIGNAL AREA : NAME->X_Axl3_Brk_Ling_1 LENGTH->8 STARTBIT :32"}
Raw_X_Axl3_Brk_Ling_1					:= _FB_CanRx_Message_221.X_Byte_4;
GVL.IIVD.X_Axl3_Brk_Ling_1.e			:= (Raw_X_Axl3_Brk_Ling_1 > 16#FD) AND (Raw_X_Axl3_Brk_Ling_1 < 16#FF);
GVL.IIVD.X_Axl3_Brk_Ling_1.na			:= (Raw_X_Axl3_Brk_Ling_1 = 16#FF);
GVL.IIVD.X_Axl3_Brk_Ling_1.RangeExcd	:= NOT ((USINT_TO_REAL(BYTE_TO_USINT(Raw_X_Axl3_Brk_Ling_1)) >= 0) AND (USINT_TO_REAL(BYTE_TO_USINT(Raw_X_Axl3_Brk_Ling_1)) <= 100));
GVL.IIVD.X_Axl3_Brk_Ling_1.v			:= NOT( GVL.IIVD.S_TmOut_Fren_balata_durumlari_0X221 OR GVL.IIVD.X_Axl3_Brk_Ling_1.RangeExcd OR GVL.IIVD.X_Axl3_Brk_Ling_1.e OR GVL.IIVD.X_Axl3_Brk_Ling_1.na) ;
GVL.IIVD.X_Axl3_Brk_Ling_1.x			:= 
(*SELECT 1 : Is data valid ?*)				SEL(GVL.IIVD.X_Axl3_Brk_Ling_1.v,
(*DEFAULT value assigment*)					0,
(*Transmission is VALID*)					USINT_TO_REAL(BYTE_TO_USINT(Raw_X_Axl3_Brk_Ling_1)));
{endregion}
{region " SIGNAL AREA : NAME->X_Axl3_Brk_Ling_2 LENGTH->8 STARTBIT :40"}
Raw_X_Axl3_Brk_Ling_2					:= _FB_CanRx_Message_221.X_Byte_5;
GVL.IIVD.X_Axl3_Brk_Ling_2.e			:= (Raw_X_Axl3_Brk_Ling_2 > 16#FD) AND (Raw_X_Axl3_Brk_Ling_2 < 16#FF);
GVL.IIVD.X_Axl3_Brk_Ling_2.na			:= (Raw_X_Axl3_Brk_Ling_2 = 16#FF);
GVL.IIVD.X_Axl3_Brk_Ling_2.RangeExcd	:= NOT ((USINT_TO_REAL(BYTE_TO_USINT(Raw_X_Axl3_Brk_Ling_2)) >= 0) AND (USINT_TO_REAL(BYTE_TO_USINT(Raw_X_Axl3_Brk_Ling_2)) <= 100));
GVL.IIVD.X_Axl3_Brk_Ling_2.v			:= NOT( GVL.IIVD.S_TmOut_Fren_balata_durumlari_0X221 OR GVL.IIVD.X_Axl3_Brk_Ling_2.RangeExcd OR GVL.IIVD.X_Axl3_Brk_Ling_2.e OR GVL.IIVD.X_Axl3_Brk_Ling_2.na) ;
GVL.IIVD.X_Axl3_Brk_Ling_2.x			:= 
(*SELECT 1 : Is data valid ?*)				SEL(GVL.IIVD.X_Axl3_Brk_Ling_2.v,
(*DEFAULT value assigment*)					0,
(*Transmission is VALID*)					USINT_TO_REAL(BYTE_TO_USINT(Raw_X_Axl3_Brk_Ling_2)));
{endregion}
{region " SIGNAL AREA : NAME->X_Axl4_Brk_Ling_1 LENGTH->8 STARTBIT :48"}
Raw_X_Axl4_Brk_Ling_1					:= _FB_CanRx_Message_221.X_Byte_6;
GVL.IIVD.X_Axl4_Brk_Ling_1.e			:= (Raw_X_Axl4_Brk_Ling_1 > 16#FD) AND (Raw_X_Axl4_Brk_Ling_1 < 16#FF);
GVL.IIVD.X_Axl4_Brk_Ling_1.na			:= (Raw_X_Axl4_Brk_Ling_1 = 16#FF);
GVL.IIVD.X_Axl4_Brk_Ling_1.RangeExcd	:= NOT ((USINT_TO_REAL(BYTE_TO_USINT(Raw_X_Axl4_Brk_Ling_1)) >= 0) AND (USINT_TO_REAL(BYTE_TO_USINT(Raw_X_Axl4_Brk_Ling_1)) <= 100));
GVL.IIVD.X_Axl4_Brk_Ling_1.v			:= NOT( GVL.IIVD.S_TmOut_Fren_balata_durumlari_0X221 OR GVL.IIVD.X_Axl4_Brk_Ling_1.RangeExcd OR GVL.IIVD.X_Axl4_Brk_Ling_1.e OR GVL.IIVD.X_Axl4_Brk_Ling_1.na) ;
GVL.IIVD.X_Axl4_Brk_Ling_1.x			:= 
(*SELECT 1 : Is data valid ?*)				SEL(GVL.IIVD.X_Axl4_Brk_Ling_1.v,
(*DEFAULT value assigment*)					0,
(*Transmission is VALID*)					USINT_TO_REAL(BYTE_TO_USINT(Raw_X_Axl4_Brk_Ling_1)));
{endregion}
{region " SIGNAL AREA : NAME->X_Axl4_Brk_Ling_2 LENGTH->8 STARTBIT :56"}
Raw_X_Axl4_Brk_Ling_2					:= _FB_CanRx_Message_221.X_Byte_7;
GVL.IIVD.X_Axl4_Brk_Ling_2.e			:= (Raw_X_Axl4_Brk_Ling_2 > 16#FD) AND (Raw_X_Axl4_Brk_Ling_2 < 16#FF);
GVL.IIVD.X_Axl4_Brk_Ling_2.na			:= (Raw_X_Axl4_Brk_Ling_2 = 16#FF);
GVL.IIVD.X_Axl4_Brk_Ling_2.RangeExcd	:= NOT ((USINT_TO_REAL(BYTE_TO_USINT(Raw_X_Axl4_Brk_Ling_2)) >= 0) AND (USINT_TO_REAL(BYTE_TO_USINT(Raw_X_Axl4_Brk_Ling_2)) <= 100));
GVL.IIVD.X_Axl4_Brk_Ling_2.v			:= NOT( GVL.IIVD.S_TmOut_Fren_balata_durumlari_0X221 OR GVL.IIVD.X_Axl4_Brk_Ling_2.RangeExcd OR GVL.IIVD.X_Axl4_Brk_Ling_2.e OR GVL.IIVD.X_Axl4_Brk_Ling_2.na) ;
GVL.IIVD.X_Axl4_Brk_Ling_2.x			:= 
(*SELECT 1 : Is data valid ?*)				SEL(GVL.IIVD.X_Axl4_Brk_Ling_2.v,
(*DEFAULT value assigment*)					0,
(*Transmission is VALID*)					USINT_TO_REAL(BYTE_TO_USINT(Raw_X_Axl4_Brk_Ling_2)));
{endregion}
{endregion}

{region " MESSAGE AREA :Fren_Basinclari- ID:222"}

_FB_CanRx_Message_Unpack_222 (	C_Enable	:= GVL.IIVD.S_CAN_Init,
    							Obj_CAN		:= ADR(GVL.IC.Obj_CAN0),
    							X_MsgID		:= 16#222,
    							Tm_MsgTmOut	:= TIME#2500MS,
    							S_Extended	:= 0,
    							S_ER_TmOut	=> GVL.IIVD.S_TmOut_Fren_Basinclari_0X222);

{region " SIGNAL AREA : NAME->S_ER_Not_Ins_Pr_Sns_Frnt_Brk LENGTH->2 STARTBIT :0"}
GVL.IIVD.S_ER_Not_Ins_Pr_Sns_Frnt_Brk.v		:= NOT GVL.IIVD.S_TmOut_Fren_Basinclari_0X222 AND NOT _FB_CanRx_Message_Unpack_222.S_Bit_1;
GVL.IIVD.S_ER_Not_Ins_Pr_Sns_Frnt_Brk.x		:= GVL.IIVD.S_ER_Not_Ins_Pr_Sns_Frnt_Brk.v AND _FB_CanRx_Message_Unpack_222.S_Bit_0;
GVL.IIVD.S_ER_Not_Ins_Pr_Sns_Frnt_Brk.e		:= _FB_CanRx_Message_Unpack_222.S_Bit_1 AND NOT _FB_CanRx_Message_Unpack_222.S_Bit_0 ;
GVL.IIVD.S_ER_Not_Ins_Pr_Sns_Frnt_Brk.na	:= _FB_CanRx_Message_Unpack_222.S_Bit_1 AND _FB_CanRx_Message_Unpack_222.S_Bit_0 ;
{endregion}
{region " SIGNAL AREA : NAME->S_ER_Not_Ins_Pr_Sns_Bwd_Brk LENGTH->2 STARTBIT :2"}
GVL.IIVD.S_ER_Not_Ins_Pr_Sns_Bwd_Brk.v		:= NOT GVL.IIVD.S_TmOut_Fren_Basinclari_0X222 AND NOT _FB_CanRx_Message_Unpack_222.S_Bit_3;
GVL.IIVD.S_ER_Not_Ins_Pr_Sns_Bwd_Brk.x		:= GVL.IIVD.S_ER_Not_Ins_Pr_Sns_Bwd_Brk.v AND _FB_CanRx_Message_Unpack_222.S_Bit_2;
GVL.IIVD.S_ER_Not_Ins_Pr_Sns_Bwd_Brk.e		:= _FB_CanRx_Message_Unpack_222.S_Bit_3 AND NOT _FB_CanRx_Message_Unpack_222.S_Bit_2 ;
GVL.IIVD.S_ER_Not_Ins_Pr_Sns_Bwd_Brk.na		:= _FB_CanRx_Message_Unpack_222.S_Bit_3 AND _FB_CanRx_Message_Unpack_222.S_Bit_2 ;
{endregion}
{region " SIGNAL AREA : NAME->S_ER_Not_Ins_Pr_Snsr_Prk_Brk LENGTH->2 STARTBIT :4"}
GVL.IIVD.S_ER_Not_Ins_Pr_Snsr_Prk_Brk.v		:= NOT GVL.IIVD.S_TmOut_Fren_Basinclari_0X222 AND NOT _FB_CanRx_Message_Unpack_222.S_Bit_5;
GVL.IIVD.S_ER_Not_Ins_Pr_Snsr_Prk_Brk.x		:= GVL.IIVD.S_ER_Not_Ins_Pr_Snsr_Prk_Brk.v AND _FB_CanRx_Message_Unpack_222.S_Bit_4;
GVL.IIVD.S_ER_Not_Ins_Pr_Snsr_Prk_Brk.e		:= _FB_CanRx_Message_Unpack_222.S_Bit_5 AND NOT _FB_CanRx_Message_Unpack_222.S_Bit_4 ;
GVL.IIVD.S_ER_Not_Ins_Pr_Snsr_Prk_Brk.na	:= _FB_CanRx_Message_Unpack_222.S_Bit_5 AND _FB_CanRx_Message_Unpack_222.S_Bit_4 ;
{endregion}
{region " SIGNAL AREA : NAME->S_ER_Not_Ins_Pr_Sns_Susp LENGTH->2 STARTBIT :6"}
GVL.IIVD.S_ER_Not_Ins_Pr_Sns_Susp_Rr.v		:= NOT GVL.IIVD.S_TmOut_Fren_Basinclari_0X222 AND NOT _FB_CanRx_Message_Unpack_222.S_Bit_7;
GVL.IIVD.S_ER_Not_Ins_Pr_Sns_Susp_Rr.x		:= GVL.IIVD.S_ER_Not_Ins_Pr_Sns_Susp_Rr.v AND _FB_CanRx_Message_Unpack_222.S_Bit_6;
GVL.IIVD.S_ER_Not_Ins_Pr_Sns_Susp_Rr.e		:= _FB_CanRx_Message_Unpack_222.S_Bit_7 AND NOT _FB_CanRx_Message_Unpack_222.S_Bit_6 ;
GVL.IIVD.S_ER_Not_Ins_Pr_Sns_Susp_Rr.na		:= _FB_CanRx_Message_Unpack_222.S_Bit_7 AND _FB_CanRx_Message_Unpack_222.S_Bit_6 ;
{endregion}
{region " SIGNAL AREA : NAME->S_ER_Not_Ins_Pr_Sns_Susp LENGTH->2 STARTBIT :8"}
GVL.IIVD.S_ER_Not_Ins_Pr_Sns_Susp_Frnt.v	:= NOT GVL.IIVD.S_TmOut_Fren_Basinclari_0X222 AND NOT _FB_CanRx_Message_Unpack_222.S_Bit_9;
GVL.IIVD.S_ER_Not_Ins_Pr_Sns_Susp_Frnt.x	:= GVL.IIVD.S_ER_Not_Ins_Pr_Sns_Susp_Frnt.v AND _FB_CanRx_Message_Unpack_222.S_Bit_8;
GVL.IIVD.S_ER_Not_Ins_Pr_Sns_Susp_Frnt.e	:= _FB_CanRx_Message_Unpack_222.S_Bit_9 AND NOT _FB_CanRx_Message_Unpack_222.S_Bit_8 ;
GVL.IIVD.S_ER_Not_Ins_Pr_Sns_Susp_Frnt.na	:= _FB_CanRx_Message_Unpack_222.S_Bit_9 AND _FB_CanRx_Message_Unpack_222.S_Bit_8 ;
{endregion}
{region " SIGNAL AREA : NAME->S_ER_Brk_Lnng LENGTH->2 STARTBIT :10"}
GVL.IIVD.S_ER_Brk_Lnng.v					:= NOT GVL.IIVD.S_TmOut_Fren_Basinclari_0X222 AND NOT _FB_CanRx_Message_Unpack_222.S_Bit_11;
GVL.IIVD.S_ER_Brk_Lnng.x					:= GVL.IIVD.S_ER_Brk_Lnng.v AND _FB_CanRx_Message_Unpack_222.S_Bit_10;
GVL.IIVD.S_ER_Brk_Lnng.e					:= _FB_CanRx_Message_Unpack_222.S_Bit_11 AND NOT _FB_CanRx_Message_Unpack_222.S_Bit_10;
GVL.IIVD.S_ER_Brk_Lnng.na					:= _FB_CanRx_Message_Unpack_222.S_Bit_11 AND _FB_CanRx_Message_Unpack_222.S_Bit_10;
{endregion}		   
{region " SIGNAL AREA : NAME->S_ER_Pin_Pr_Air LENGTH->2 STARTBIT :12"}
GVL.IIVD.S_ER_Pin_Pr_Air.v					:= NOT GVL.IIVD.S_TmOut_Fren_Basinclari_0X222 AND NOT _FB_CanRx_Message_Unpack_222.S_Bit_13;
GVL.IIVD.S_ER_Pin_Pr_Air.x					:= GVL.IIVD.S_ER_Pin_Pr_Air.v AND _FB_CanRx_Message_Unpack_222.S_Bit_12;
GVL.IIVD.S_ER_Pin_Pr_Air.e					:= _FB_Canrx_message_unpack_222.S_Bit_13 AND NOT _FB_Canrx_message_unpack_222.S_Bit_12;
GVL.IIVD.S_ER_Pin_Pr_Air.na					:= _FB_Canrx_message_unpack_222.S_Bit_13 AND _FB_CanRx_Message_Unpack_222.S_Bit_12;
{endregion}
{region " SIGNAL AREA : NAME->X_Pr_Air_Tank_Brk_Bwd LENGTH->8 STARTBIT :16"}
Raw_X_Pr_Air_Tank_Brk_Bwd					:= _FB_CanRx_Message_Unpack_222.X_Byte_2;
GVL.IIVD.X_Pr_Air_Tank_Brk_Bwd.e			:= (Raw_X_Pr_Air_Tank_Brk_Bwd > 16#FD) AND (Raw_X_Pr_Air_Tank_Brk_Bwd < 16#FF);
GVL.IIVD.X_Pr_Air_Tank_Brk_Bwd.na			:= (Raw_X_Pr_Air_Tank_Brk_Bwd = 16#FF);
GVL.IIVD.X_Pr_Air_Tank_Brk_Bwd.RangeExcd	:= NOT ((USINT_TO_REAL(BYTE_TO_USINT(Raw_X_Pr_Air_Tank_Brk_Bwd))*0.05 >= 0) AND (USINT_TO_REAL(BYTE_TO_USINT(Raw_X_Pr_Air_Tank_Brk_Bwd))*0.05 <= 12.5));
GVL.IIVD.X_Pr_Air_Tank_Brk_Bwd.v			:= NOT( GVL.IIVD.S_TmOut_Fren_Basinclari_0X222 OR GVL.IIVD.X_Pr_Air_Tank_Brk_Bwd.RangeExcd OR GVL.IIVD.X_Pr_Air_Tank_Brk_Bwd.e OR GVL.IIVD.X_Pr_Air_Tank_Brk_Bwd.na) ;
GVL.IIVD.X_Pr_Air_Tank_Brk_Bwd.x			:= 
(*SELECT 1 : Is data valid ?*)					SEL(GVL.IIVD.X_Pr_Air_Tank_Brk_Bwd.v,
(*DEFAULT value assigment*)						0,
(*Transmission is VALID*)						USINT_TO_REAL(BYTE_TO_USINT(Raw_X_Pr_Air_Tank_Brk_Bwd))*0.05);
{endregion}
{region " SIGNAL AREA : NAME->X_Pr_Air_Tank_Brk_Frnt LENGTH->8 STARTBIT :24"}
Raw_X_Pr_Air_Tank_Brk_Frnt					:= _FB_CanRx_Message_Unpack_222.X_Byte_3;
GVL.IIVD.X_Pr_Air_Tank_Brk_Frnt.e			:= (Raw_X_Pr_Air_Tank_Brk_Frnt > 16#FD) AND (Raw_X_Pr_Air_Tank_Brk_Frnt < 16#FF);
GVL.IIVD.X_Pr_Air_Tank_Brk_Frnt.na			:= (Raw_X_Pr_Air_Tank_Brk_Frnt = 16#FF);
GVL.IIVD.X_Pr_Air_Tank_Brk_Frnt.RangeExcd	:= NOT ((USINT_TO_REAL(BYTE_TO_USINT(Raw_X_Pr_Air_Tank_Brk_Frnt))*0.05 >= 0) AND (USINT_TO_REAL(BYTE_TO_USINT(Raw_X_Pr_Air_Tank_Brk_Frnt))*0.05 <= 12.5));
GVL.IIVD.X_Pr_Air_Tank_Brk_Frnt.v			:= NOT( GVL.IIVD.S_TmOut_Fren_Basinclari_0X222 OR GVL.IIVD.X_Pr_Air_Tank_Brk_Frnt.RangeExcd OR GVL.IIVD.X_Pr_Air_Tank_Brk_Frnt.e OR GVL.IIVD.X_Pr_Air_Tank_Brk_Frnt.na) ;
GVL.IIVD.X_Pr_Air_Tank_Brk_Frnt.x			:= 
(*SELECT 1 : Is data valid ?*)					SEL(GVL.IIVD.X_Pr_Air_Tank_Brk_Frnt.v,
(*DEFAULT value assigment*)						0,
(*Transmission is VALID*)						USINT_TO_REAL(BYTE_TO_USINT(Raw_X_Pr_Air_Tank_Brk_Frnt))*0.05);
{endregion}
{region " SIGNAL AREA : NAME->X_Pr_Air_Tank_Brk_Prk LENGTH->8 STARTBIT :32"}
Raw_X_Pr_Air_Tank_Brk_Prk					:= _FB_CanRx_Message_Unpack_222.X_Byte_4;
GVL.IIVD.X_Pr_Air_Tank_Brk_Prk.e			:= (Raw_X_Pr_Air_Tank_Brk_Prk > 16#FD) AND (Raw_X_Pr_Air_Tank_Brk_Prk < 16#FF);
GVL.IIVD.X_Pr_Air_Tank_Brk_Prk.na			:= (Raw_X_Pr_Air_Tank_Brk_Prk = 16#FF);
GVL.IIVD.X_Pr_Air_Tank_Brk_Prk.RangeExcd	:= NOT ((USINT_TO_REAL(BYTE_TO_USINT(Raw_X_Pr_Air_Tank_Brk_Prk))*0.05 >= 0) AND (USINT_TO_REAL(BYTE_TO_USINT(Raw_X_Pr_Air_Tank_Brk_Prk))*0.05 <= 12.5));
GVL.IIVD.X_Pr_Air_Tank_Brk_Prk.v			:= NOT( GVL.IIVD.S_TmOut_Fren_Basinclari_0X222 OR GVL.IIVD.X_Pr_Air_Tank_Brk_Prk.RangeExcd OR GVL.IIVD.X_Pr_Air_Tank_Brk_Prk.e OR GVL.IIVD.X_Pr_Air_Tank_Brk_Prk.na) ;
GVL.IIVD.X_Pr_Air_Tank_Brk_Prk.x			:= 
(*SELECT 1 : Is data valid ?*)					SEL(GVL.IIVD.X_Pr_Air_Tank_Brk_Prk.v,
(*DEFAULT value assigment*)						0,
(*Transmission is VALID*)						USINT_TO_REAL(BYTE_TO_USINT(Raw_X_Pr_Air_Tank_Brk_Prk))*0.05);
{endregion}
{region " SIGNAL AREA : NAME->X_Pr_Air_Tank_Susp LENGTH->8 STARTBIT :40"}
Raw_X_Pr_Air_Tank_Susp_Rr					:= _FB_CanRx_Message_Unpack_222.X_Byte_5;
GVL.IIVD.X_Pr_Air_Tank_Susp_Rr.e			:= (Raw_X_Pr_Air_Tank_Susp_Rr > 16#FD) AND (Raw_X_Pr_Air_Tank_Susp_Rr < 16#FF);
GVL.IIVD.X_Pr_Air_Tank_Susp_Rr.na			:= (Raw_X_Pr_Air_Tank_Susp_Rr = 16#FF);
GVL.IIVD.X_Pr_Air_Tank_Susp_Rr.RangeExcd	:= NOT ((USINT_TO_REAL(BYTE_TO_USINT(Raw_X_Pr_Air_Tank_Susp_Rr))*0.05 >= 0) AND (USINT_TO_REAL(BYTE_TO_USINT(Raw_X_Pr_Air_Tank_Susp_Rr))*0.05 <= 12.5));
GVL.IIVD.X_Pr_Air_Tank_Susp_Rr.v			:= NOT( GVL.IIVD.S_TmOut_Fren_Basinclari_0X222 OR GVL.IIVD.X_Pr_Air_Tank_Susp_Rr.RangeExcd OR GVL.IIVD.X_Pr_Air_Tank_Susp_Rr.e OR GVL.IIVD.X_Pr_Air_Tank_Susp_Rr.na) ;
GVL.IIVD.X_Pr_Air_Tank_Susp_Rr.x			:= 
(*SELECT 1 : Is data valid ?*)					SEL(GVL.IIVD.X_Pr_Air_Tank_Susp_Rr.v,
(*DEFAULT value assigment*)						0,
(*Transmission is VALID*)						USINT_TO_REAL(BYTE_TO_USINT(Raw_X_Pr_Air_Tank_Susp_Rr))*0.05);
{endregion}
{region " SIGNAL AREA : NAME->X_Pr_Air_Tank_Susp LENGTH->8 STARTBIT :48"}
Raw_X_Pr_Air_Tank_Susp_Frnt					:= _FB_CanRx_Message_Unpack_222.X_Byte_5;
GVL.IIVD.X_Pr_Air_Tank_Susp_Frnt.e			:= (Raw_X_Pr_Air_Tank_Susp_Frnt > 16#FD) AND (Raw_X_Pr_Air_Tank_Susp_Frnt < 16#FF);
GVL.IIVD.X_Pr_Air_Tank_Susp_Frnt.na			:= (Raw_X_Pr_Air_Tank_Susp_Frnt = 16#FF);
GVL.IIVD.X_Pr_Air_Tank_Susp_Frnt.RangeExcd	:= NOT ((USINT_TO_REAL(BYTE_TO_USINT(Raw_X_Pr_Air_Tank_Susp_Frnt))*0.05 >= 0) AND (USINT_TO_REAL(BYTE_TO_USINT(Raw_X_Pr_Air_Tank_Susp_Frnt))*0.05 <= 12.5));
GVL.IIVD.X_Pr_Air_Tank_Susp_Frnt.v			:= NOT( GVL.IIVD.S_TmOut_Fren_Basinclari_0X222 OR GVL.IIVD.X_Pr_Air_Tank_Susp_Frnt.RangeExcd OR GVL.IIVD.X_Pr_Air_Tank_Susp_Frnt.e OR GVL.IIVD.X_Pr_Air_Tank_Susp_Frnt.na) ;
GVL.IIVD.X_Pr_Air_Tank_Susp_Frnt.x			:= 
(*SELECT 1 : Is data valid ?*)					SEL(GVL.IIVD.X_Pr_Air_Tank_Susp_Frnt.v,
(*DEFAULT value assigment*)						0,
(*Transmission is VALID*)						USINT_TO_REAL(BYTE_TO_USINT(Raw_X_Pr_Air_Tank_Susp_Frnt))*0.05);
{endregion}
{endregion}
{region " MESSAGE AREA :Lastik_Basinclari_1- ID:223"}

_FB_CanRx_Message_223 (		C_Enable	:= GVL.IIVD.S_CAN_Init,
     						Obj_CAN		:= ADR(GVL.IC.Obj_CAN0),
     						X_MsgID		:= 16#223,
     						Tm_MsgTmOut	:= TIME#2500MS,
     						S_Extended	:= 0,
     						S_ER_TmOut	=> GVL.IIVD.S_TmOut_Lastik_Basinclari_1_0X223);

{region " SIGNAL AREA : NAME->X_Pr_Axl1_Wh1 LENGTH->8 STARTBIT :0"}
Raw_X_Pr_Axl1_Wh1						:= _FB_CanRx_Message_223.X_Byte_0;
GVL.IIVD.X_Pr_Axl1_Wh1.e				:= (Raw_X_Pr_Axl1_Wh1 > 16#FD) AND (Raw_X_Pr_Axl1_Wh1 < 16#FF);
GVL.IIVD.X_Pr_Axl1_Wh1.na				:= (Raw_X_Pr_Axl1_Wh1 = 16#FF);
GVL.IIVD.X_Pr_Axl1_Wh1.RangeExcd		:= NOT ((USINT_TO_REAL(BYTE_TO_USINT(Raw_X_Pr_Axl1_Wh1)) >= 0) AND (USINT_TO_REAL(BYTE_TO_USINT(Raw_X_Pr_Axl1_Wh1)) <= 250));
GVL.IIVD.X_Pr_Axl1_Wh1.v				:= NOT( GVL.IIVD.S_TmOut_Lastik_Basinclari_1_0X223 OR GVL.IIVD.X_Pr_Axl1_Wh1.RangeExcd OR GVL.IIVD.X_Pr_Axl1_Wh1.e OR GVL.IIVD.X_Pr_Axl1_Wh1.na) ;
GVL.IIVD.X_Pr_Axl1_Wh1.x				:= 
(*SELECT 1 : Is data valid ?*)				SEL(GVL.IIVD.X_Pr_Axl1_Wh1.v,
(*DEFAULT value assigment*)					0,
(*Transmission is VALID*)					USINT_TO_REAL(BYTE_TO_USINT(Raw_X_Pr_Axl1_Wh1)));
{endregion}
{region " SIGNAL AREA : NAME->X_Pr_Axl1_Wh2 LENGTH->8 STARTBIT :8"}
Raw_X_Pr_Axl1_Wh2		:= _FB_CanRx_Message_223.X_Byte_1;
GVL.IIVD.X_Pr_Axl1_Wh2.e				:= (Raw_X_Pr_Axl1_Wh2 > 16#FD) AND (Raw_X_Pr_Axl1_Wh2 < 16#FF);
GVL.IIVD.X_Pr_Axl1_Wh2.na				:= (Raw_X_Pr_Axl1_Wh2 = 16#FF);
GVL.IIVD.X_Pr_Axl1_Wh2.RangeExcd		:= NOT ((USINT_TO_REAL(BYTE_TO_USINT(Raw_X_Pr_Axl1_Wh2)) >= 0) AND (USINT_TO_REAL(BYTE_TO_USINT(Raw_X_Pr_Axl1_Wh2)) <= 250));
GVL.IIVD.X_Pr_Axl1_Wh2.v				:= NOT( GVL.IIVD.S_TmOut_Lastik_Basinclari_1_0X223 OR GVL.IIVD.X_Pr_Axl1_Wh2.RangeExcd OR GVL.IIVD.X_Pr_Axl1_Wh2.e OR GVL.IIVD.X_Pr_Axl1_Wh2.na) ;
GVL.IIVD.X_Pr_Axl1_Wh2.x				:= 
(*SELECT 1 : Is data valid ?*)				SEL(GVL.IIVD.X_Pr_Axl1_Wh2.v,
(*DEFAULT value assigment*)					0,
(*Transmission is VALID*)					USINT_TO_REAL(BYTE_TO_USINT(Raw_X_Pr_Axl1_Wh2)));
{endregion}
{region " SIGNAL AREA : NAME->X_Pr_Axl2_Wh1 LENGTH->8 STARTBIT :16"}
Raw_X_Pr_Axl2_Wh1						:= _FB_CanRx_Message_223.X_Byte_2;
GVL.IIVD.X_Pr_Axl2_Wh1.e				:= (Raw_X_Pr_Axl2_Wh1 > 16#FD) AND (Raw_X_Pr_Axl2_Wh1 < 16#FF);
GVL.IIVD.X_Pr_Axl2_Wh1.na				:= (Raw_X_Pr_Axl2_Wh1 = 16#FF);
GVL.IIVD.X_Pr_Axl2_Wh1.RangeExcd		:= NOT ((USINT_TO_REAL(BYTE_TO_USINT(Raw_X_Pr_Axl2_Wh1)) >= 0) AND (USINT_TO_REAL(BYTE_TO_USINT(Raw_X_Pr_Axl2_Wh1)) <= 250));
GVL.IIVD.X_Pr_Axl2_Wh1.v				:= NOT( GVL.IIVD.S_TmOut_Lastik_Basinclari_1_0X223 OR GVL.IIVD.X_Pr_Axl2_Wh1.RangeExcd OR GVL.IIVD.X_Pr_Axl2_Wh1.e OR GVL.IIVD.X_Pr_Axl2_Wh1.na) ;
GVL.IIVD.X_Pr_Axl2_Wh1.x				:= 
(*SELECT 1 : Is data valid ?*)				SEL(GVL.IIVD.X_Pr_Axl2_Wh1.v,
(*DEFAULT value assigment*)					0,
(*Transmission is VALID*)					USINT_TO_REAL(BYTE_TO_USINT(Raw_X_Pr_Axl2_Wh1)));
{endregion}
{region " SIGNAL AREA : NAME->X_Pr_Axl2_Wh2 LENGTH->8 STARTBIT :24"}
Raw_X_Pr_Axl2_Wh2						:= _FB_CanRx_Message_223.X_Byte_3;
GVL.IIVD.X_Pr_Axl2_Wh2.e				:= (Raw_X_Pr_Axl2_Wh2 > 16#FD) AND (Raw_X_Pr_Axl2_Wh2 < 16#FF);
GVL.IIVD.X_Pr_Axl2_Wh2.na				:= (Raw_X_Pr_Axl2_Wh2 = 16#FF);
GVL.IIVD.X_Pr_Axl2_Wh2.RangeExcd		:= NOT ((USINT_TO_REAL(BYTE_TO_USINT(Raw_X_Pr_Axl2_Wh2)) >= 0) AND (USINT_TO_REAL(BYTE_TO_USINT(Raw_X_Pr_Axl2_Wh2)) <= 250));
GVL.IIVD.X_Pr_Axl2_Wh2.v				:= NOT( GVL.IIVD.S_TmOut_Lastik_Basinclari_1_0X223 OR GVL.IIVD.X_Pr_Axl2_Wh2.RangeExcd OR GVL.IIVD.X_Pr_Axl2_Wh2.e OR GVL.IIVD.X_Pr_Axl2_Wh2.na) ;
GVL.IIVD.X_Pr_Axl2_Wh2.x				:= 
(*SELECT 1 : Is data valid ?*)				SEL(GVL.IIVD.X_Pr_Axl2_Wh2.v,
(*DEFAULT value assigment*)					0,
(*Transmission is VALID*)					USINT_TO_REAL(BYTE_TO_USINT(Raw_X_Pr_Axl2_Wh2)));
{endregion}
{region " SIGNAL AREA : NAME->X_Pr_Axl2_Wh3 LENGTH->8 STARTBIT :32"}
Raw_X_Pr_Axl2_Wh3						:= _FB_CanRx_Message_223.X_Byte_4;
GVL.IIVD.X_Pr_Axl2_Wh3.e				:= (Raw_X_Pr_Axl2_Wh3 > 16#FD) AND (Raw_X_Pr_Axl2_Wh3 < 16#FF);
GVL.IIVD.X_Pr_Axl2_Wh3.na				:= (Raw_X_Pr_Axl2_Wh3 = 16#FF);
GVL.IIVD.X_Pr_Axl2_Wh3.RangeExcd		:= NOT ((USINT_TO_REAL(BYTE_TO_USINT(Raw_X_Pr_Axl2_Wh3)) >= 0) AND (USINT_TO_REAL(BYTE_TO_USINT(Raw_X_Pr_Axl2_Wh3)) <= 250));
GVL.IIVD.X_Pr_Axl2_Wh3.v				:= NOT( GVL.IIVD.S_TmOut_Lastik_Basinclari_1_0X223 OR GVL.IIVD.X_Pr_Axl2_Wh3.RangeExcd OR GVL.IIVD.X_Pr_Axl2_Wh3.e OR GVL.IIVD.X_Pr_Axl2_Wh3.na) ;
GVL.IIVD.X_Pr_Axl2_Wh3.x				:= 
(*SELECT 1 : Is data valid ?*)				SEL(GVL.IIVD.X_Pr_Axl2_Wh3.v,
(*DEFAULT value assigment*)					0,
(*Transmission is VALID*)					USINT_TO_REAL(BYTE_TO_USINT(Raw_X_Pr_Axl2_Wh3)));
{endregion}
{region " SIGNAL AREA : NAME->X_Pr_Axl2_Wh4 LENGTH->8 STARTBIT :40"}
Raw_X_Pr_Axl2_Wh4						:= _FB_CanRx_Message_223.X_Byte_5;
GVL.IIVD.X_Pr_Axl2_Wh4.e				:= (Raw_X_Pr_Axl2_Wh4 > 16#FD) AND (Raw_X_Pr_Axl2_Wh4 < 16#FF);
GVL.IIVD.X_Pr_Axl2_Wh4.na				:= (Raw_X_Pr_Axl2_Wh4 = 16#FF);
GVL.IIVD.X_Pr_Axl2_Wh4.RangeExcd		:= NOT ((USINT_TO_REAL(BYTE_TO_USINT(Raw_X_Pr_Axl2_Wh4)) >= 0) AND (USINT_TO_REAL(BYTE_TO_USINT(Raw_X_Pr_Axl2_Wh4)) <= 250));
GVL.IIVD.X_Pr_Axl2_Wh4.v				:= NOT( GVL.IIVD.S_TmOut_Lastik_Basinclari_1_0X223 OR GVL.IIVD.X_Pr_Axl2_Wh4.RangeExcd OR GVL.IIVD.X_Pr_Axl2_Wh4.e OR GVL.IIVD.X_Pr_Axl2_Wh4.na) ;
GVL.IIVD.X_Pr_Axl2_Wh4.x				:= 
(*SELECT 1 : Is data valid ?*)				SEL(GVL.IIVD.X_Pr_Axl2_Wh4.v,
(*DEFAULT value assigment*)					0,
(*Transmission is VALID*)					USINT_TO_REAL(BYTE_TO_USINT(Raw_X_Pr_Axl2_Wh4)));
{endregion}
{endregion}

{region " MESSAGE AREA :Lastik_Basinclari_2- ID:224"}

_FB_CanRx_Message_224 (		C_Enable	:= GVL.IIVD.S_CAN_Init,
     						Obj_CAN		:= ADR(GVL.IC.Obj_CAN0),
     						X_MsgID		:= 16#224,
     						Tm_MsgTmOut	:= TIME#2500MS,
     						S_Extended	:= 0,
     						S_ER_TmOut	=> GVL.IIVD.S_TmOut_Lastik_Basinclari_2_0X224);

